// TIA Portal V17 export
// export: Created 2023-02-13T11:16:53.9943503Z, ExportSetting WithDefaults, DisplayName Totally Integrated Automation Portal, DisplayVersion V17, DisplayName TIA Portal Openness, DisplayVersion V17, DisplayName TIA Portal Teamcenter Gateway, DisplayVersion V17, DisplayName TIA Portal Version Control Interface, DisplayVersion V17, DisplayName SINAMICS Startdrive Advanced, DisplayVersion V17, DisplayName SINAMICS Startdrive G130, G150, S120, S150, SINAMICS MV, S210, DisplayVersion V17, DisplayName SINAMICS Startdrive G110M, G120, G120C, G120D, G120P, G115D, DisplayVersion V17, DisplayName STEP 7 Professional, DisplayVersion V17, DisplayName STEP 7 Safety, DisplayVersion V17, DisplayName WinCC Professional, DisplayVersion V17
FUNCTION "Blending" : Void   // FC8, LAD
{ S7_Optimized_Access := 'TRUE' }
VERSION : 0.1
// stored: AutoNumber true, IsIECCheckEnabled false, SetENOAutomatically false, UDAEnableTagReadback false
   VAR_TEMP   // added for the SCL form of the ladder/FBD networks
      _w1 : Bool;
   END_VAR
BEGIN

REGION Network 1
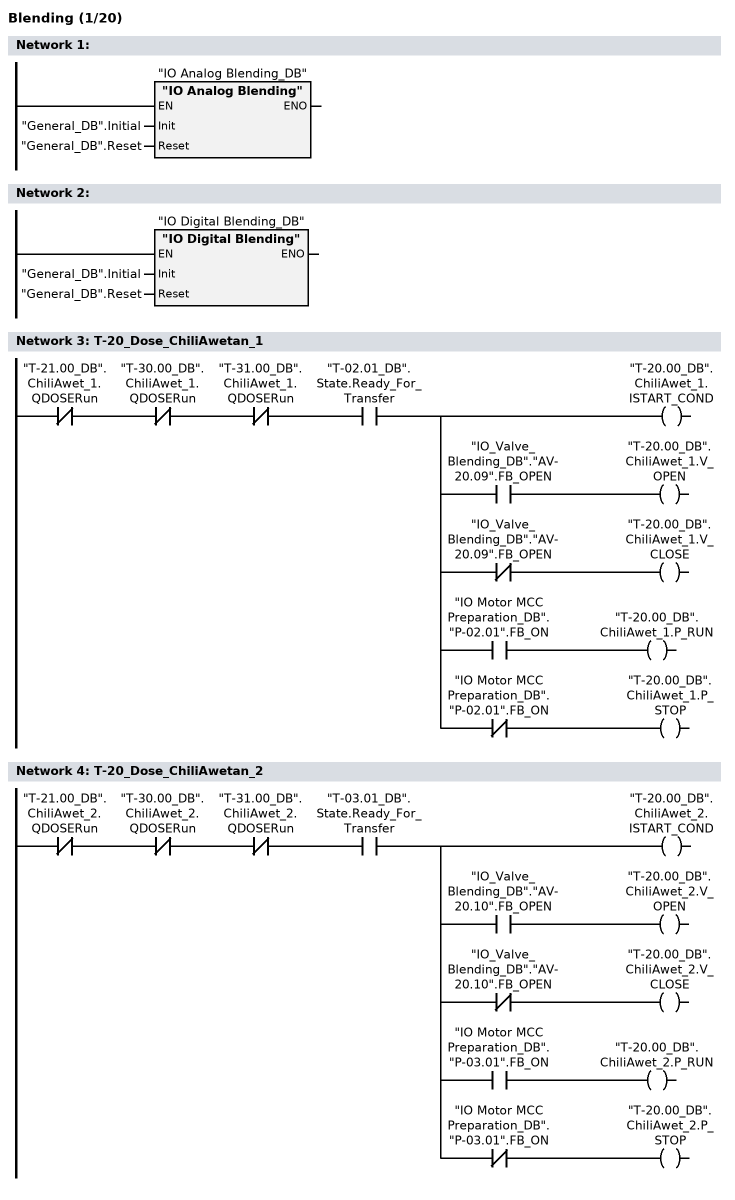
   RUNG wire#powerrail
      "IO Analog Blending_DB"(Init := "General_DB".Initial, Reset := "General_DB".Reset)
   END_RUNG
   // the same network as SCL:
   "IO Analog Blending_DB"(Init := "General_DB".Initial, Reset := "General_DB".Reset);   // "IO Analog Blending"
END_REGION

REGION Network 2
   RUNG wire#powerrail
      "IO Digital Blending_DB"(Init := "General_DB".Initial, Reset := "General_DB".Reset)
   END_RUNG
   // the same network as SCL:
   "IO Digital Blending_DB"(Init := "General_DB".Initial, Reset := "General_DB".Reset);   // "IO Digital Blending"
END_REGION

REGION Network 3: T-20_Dose_ChiliAwetan_1
   RUNG wire#powerrail
      I_Contact( "T-21.00_DB".ChiliAwet_1.QDOSERun )
      I_Contact( "T-30.00_DB".ChiliAwet_1.QDOSERun )
      I_Contact( "T-31.00_DB".ChiliAwet_1.QDOSERun )
      Contact( "T-02.01_DB".State.Ready_For_Transfer )
      wire#w1
      Coil( "T-20.00_DB".ChiliAwet_1.ISTART_COND )
   END_RUNG
   RUNG wire#w1
      Contact( "IO_Valve_Blending_DB"."AV-20.09".FB_OPEN )
      Coil( "T-20.00_DB".ChiliAwet_1.V_OPEN )
   END_RUNG
   RUNG wire#w1
      I_Contact( "IO_Valve_Blending_DB"."AV-20.09".FB_OPEN )
      Coil( "T-20.00_DB".ChiliAwet_1.V_CLOSE )
   END_RUNG
   RUNG wire#w1
      Contact( "IO Motor MCC Preparation_DB"."P-02.01".FB_ON )
      Coil( "T-20.00_DB".ChiliAwet_1.P_RUN )
   END_RUNG
   RUNG wire#w1
      I_Contact( "IO Motor MCC Preparation_DB"."P-02.01".FB_ON )
      Coil( "T-20.00_DB".ChiliAwet_1.P_STOP )
   END_RUNG
   // the same network as SCL:
   "T-20.00_DB".ChiliAwet_1.ISTART_COND := NOT "T-21.00_DB".ChiliAwet_1.QDOSERun AND NOT "T-30.00_DB".ChiliAwet_1.QDOSERun AND NOT "T-31.00_DB".ChiliAwet_1.QDOSERun AND "T-02.01_DB".State.Ready_For_Transfer;
   "T-20.00_DB".ChiliAwet_1.V_OPEN := "T-20.00_DB".ChiliAwet_1.ISTART_COND AND "IO_Valve_Blending_DB"."AV-20.09".FB_OPEN;
   "T-20.00_DB".ChiliAwet_1.V_CLOSE := "T-20.00_DB".ChiliAwet_1.ISTART_COND AND NOT "IO_Valve_Blending_DB"."AV-20.09".FB_OPEN;
   "T-20.00_DB".ChiliAwet_1.P_RUN := "T-20.00_DB".ChiliAwet_1.ISTART_COND AND "IO Motor MCC Preparation_DB"."P-02.01".FB_ON;
   "T-20.00_DB".ChiliAwet_1.P_STOP := "T-20.00_DB".ChiliAwet_1.ISTART_COND AND NOT "IO Motor MCC Preparation_DB"."P-02.01".FB_ON;
END_REGION

REGION Network 4: T-20_Dose_ChiliAwetan_2
   RUNG wire#powerrail
      I_Contact( "T-21.00_DB".ChiliAwet_2.QDOSERun )
      I_Contact( "T-30.00_DB".ChiliAwet_2.QDOSERun )
      I_Contact( "T-31.00_DB".ChiliAwet_2.QDOSERun )
      Contact( "T-03.01_DB".State.Ready_For_Transfer )
      wire#w1
      Coil( "T-20.00_DB".ChiliAwet_2.ISTART_COND )
   END_RUNG
   RUNG wire#w1
      Contact( "IO_Valve_Blending_DB"."AV-20.10".FB_OPEN )
      Coil( "T-20.00_DB".ChiliAwet_2.V_OPEN )
   END_RUNG
   RUNG wire#w1
      I_Contact( "IO_Valve_Blending_DB"."AV-20.10".FB_OPEN )
      Coil( "T-20.00_DB".ChiliAwet_2.V_CLOSE )
   END_RUNG
   RUNG wire#w1
      Contact( "IO Motor MCC Preparation_DB"."P-03.01".FB_ON )
      Coil( "T-20.00_DB".ChiliAwet_2.P_RUN )
   END_RUNG
   RUNG wire#w1
      I_Contact( "IO Motor MCC Preparation_DB"."P-03.01".FB_ON )
      Coil( "T-20.00_DB".ChiliAwet_2.P_STOP )
   END_RUNG
   // the same network as SCL:
   "T-20.00_DB".ChiliAwet_2.ISTART_COND := NOT "T-21.00_DB".ChiliAwet_2.QDOSERun AND NOT "T-30.00_DB".ChiliAwet_2.QDOSERun AND NOT "T-31.00_DB".ChiliAwet_2.QDOSERun AND "T-03.01_DB".State.Ready_For_Transfer;
   "T-20.00_DB".ChiliAwet_2.V_OPEN := "T-20.00_DB".ChiliAwet_2.ISTART_COND AND "IO_Valve_Blending_DB"."AV-20.10".FB_OPEN;
   "T-20.00_DB".ChiliAwet_2.V_CLOSE := "T-20.00_DB".ChiliAwet_2.ISTART_COND AND NOT "IO_Valve_Blending_DB"."AV-20.10".FB_OPEN;
   "T-20.00_DB".ChiliAwet_2.P_RUN := "T-20.00_DB".ChiliAwet_2.ISTART_COND AND "IO Motor MCC Preparation_DB"."P-03.01".FB_ON;
   "T-20.00_DB".ChiliAwet_2.P_STOP := "T-20.00_DB".ChiliAwet_2.ISTART_COND AND NOT "IO Motor MCC Preparation_DB"."P-03.01".FB_ON;
END_REGION

REGION Network 5: T-20_Dose_ChiliAwetan_3
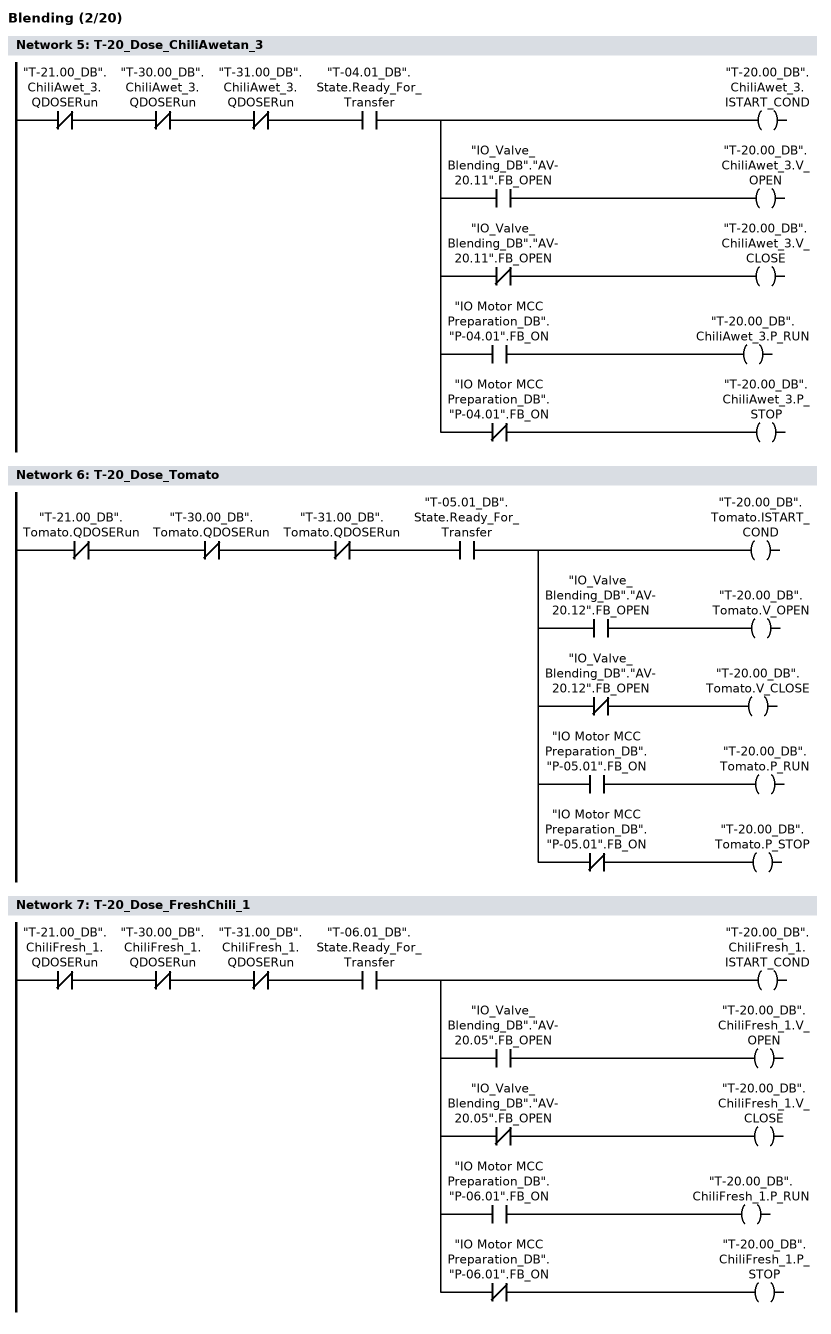
   RUNG wire#powerrail
      I_Contact( "T-21.00_DB".ChiliAwet_3.QDOSERun )
      I_Contact( "T-30.00_DB".ChiliAwet_3.QDOSERun )
      I_Contact( "T-31.00_DB".ChiliAwet_3.QDOSERun )
      Contact( "T-04.01_DB".State.Ready_For_Transfer )
      wire#w1
      Coil( "T-20.00_DB".ChiliAwet_3.ISTART_COND )
   END_RUNG
   RUNG wire#w1
      Contact( "IO_Valve_Blending_DB"."AV-20.11".FB_OPEN )
      Coil( "T-20.00_DB".ChiliAwet_3.V_OPEN )
   END_RUNG
   RUNG wire#w1
      I_Contact( "IO_Valve_Blending_DB"."AV-20.11".FB_OPEN )
      Coil( "T-20.00_DB".ChiliAwet_3.V_CLOSE )
   END_RUNG
   RUNG wire#w1
      Contact( "IO Motor MCC Preparation_DB"."P-04.01".FB_ON )
      Coil( "T-20.00_DB".ChiliAwet_3.P_RUN )
   END_RUNG
   RUNG wire#w1
      I_Contact( "IO Motor MCC Preparation_DB"."P-04.01".FB_ON )
      Coil( "T-20.00_DB".ChiliAwet_3.P_STOP )
   END_RUNG
   // the same network as SCL:
   "T-20.00_DB".ChiliAwet_3.ISTART_COND := NOT "T-21.00_DB".ChiliAwet_3.QDOSERun AND NOT "T-30.00_DB".ChiliAwet_3.QDOSERun AND NOT "T-31.00_DB".ChiliAwet_3.QDOSERun AND "T-04.01_DB".State.Ready_For_Transfer;
   "T-20.00_DB".ChiliAwet_3.V_OPEN := "T-20.00_DB".ChiliAwet_3.ISTART_COND AND "IO_Valve_Blending_DB"."AV-20.11".FB_OPEN;
   "T-20.00_DB".ChiliAwet_3.V_CLOSE := "T-20.00_DB".ChiliAwet_3.ISTART_COND AND NOT "IO_Valve_Blending_DB"."AV-20.11".FB_OPEN;
   "T-20.00_DB".ChiliAwet_3.P_RUN := "T-20.00_DB".ChiliAwet_3.ISTART_COND AND "IO Motor MCC Preparation_DB"."P-04.01".FB_ON;
   "T-20.00_DB".ChiliAwet_3.P_STOP := "T-20.00_DB".ChiliAwet_3.ISTART_COND AND NOT "IO Motor MCC Preparation_DB"."P-04.01".FB_ON;
END_REGION

REGION Network 6: T-20_Dose_Tomato
   RUNG wire#powerrail
      I_Contact( "T-21.00_DB".Tomato.QDOSERun )
      I_Contact( "T-30.00_DB".Tomato.QDOSERun )
      I_Contact( "T-31.00_DB".Tomato.QDOSERun )
      Contact( "T-05.01_DB".State.Ready_For_Transfer )
      wire#w1
      Coil( "T-20.00_DB".Tomato.ISTART_COND )
   END_RUNG
   RUNG wire#w1
      Contact( "IO_Valve_Blending_DB"."AV-20.12".FB_OPEN )
      Coil( "T-20.00_DB".Tomato.V_OPEN )
   END_RUNG
   RUNG wire#w1
      I_Contact( "IO_Valve_Blending_DB"."AV-20.12".FB_OPEN )
      Coil( "T-20.00_DB".Tomato.V_CLOSE )
   END_RUNG
   RUNG wire#w1
      Contact( "IO Motor MCC Preparation_DB"."P-05.01".FB_ON )
      Coil( "T-20.00_DB".Tomato.P_RUN )
   END_RUNG
   RUNG wire#w1
      I_Contact( "IO Motor MCC Preparation_DB"."P-05.01".FB_ON )
      Coil( "T-20.00_DB".Tomato.P_STOP )
   END_RUNG
   // the same network as SCL:
   "T-20.00_DB".Tomato.ISTART_COND := NOT "T-21.00_DB".Tomato.QDOSERun AND NOT "T-30.00_DB".Tomato.QDOSERun AND NOT "T-31.00_DB".Tomato.QDOSERun AND "T-05.01_DB".State.Ready_For_Transfer;
   "T-20.00_DB".Tomato.V_OPEN := "T-20.00_DB".Tomato.ISTART_COND AND "IO_Valve_Blending_DB"."AV-20.12".FB_OPEN;
   "T-20.00_DB".Tomato.V_CLOSE := "T-20.00_DB".Tomato.ISTART_COND AND NOT "IO_Valve_Blending_DB"."AV-20.12".FB_OPEN;
   "T-20.00_DB".Tomato.P_RUN := "T-20.00_DB".Tomato.ISTART_COND AND "IO Motor MCC Preparation_DB"."P-05.01".FB_ON;
   "T-20.00_DB".Tomato.P_STOP := "T-20.00_DB".Tomato.ISTART_COND AND NOT "IO Motor MCC Preparation_DB"."P-05.01".FB_ON;
END_REGION

REGION Network 7: T-20_Dose_FreshChili_1
   RUNG wire#powerrail
      I_Contact( "T-21.00_DB".ChiliFresh_1.QDOSERun )
      I_Contact( "T-30.00_DB".ChiliFresh_1.QDOSERun )
      I_Contact( "T-31.00_DB".ChiliFresh_1.QDOSERun )
      Contact( "T-06.01_DB".State.Ready_For_Transfer )
      wire#w1
      Coil( "T-20.00_DB".ChiliFresh_1.ISTART_COND )
   END_RUNG
   RUNG wire#w1
      Contact( "IO_Valve_Blending_DB"."AV-20.05".FB_OPEN )
      Coil( "T-20.00_DB".ChiliFresh_1.V_OPEN )
   END_RUNG
   RUNG wire#w1
      I_Contact( "IO_Valve_Blending_DB"."AV-20.05".FB_OPEN )
      Coil( "T-20.00_DB".ChiliFresh_1.V_CLOSE )
   END_RUNG
   RUNG wire#w1
      Contact( "IO Motor MCC Preparation_DB"."P-06.01".FB_ON )
      Coil( "T-20.00_DB".ChiliFresh_1.P_RUN )
   END_RUNG
   RUNG wire#w1
      I_Contact( "IO Motor MCC Preparation_DB"."P-06.01".FB_ON )
      Coil( "T-20.00_DB".ChiliFresh_1.P_STOP )
   END_RUNG
   // the same network as SCL:
   "T-20.00_DB".ChiliFresh_1.ISTART_COND := NOT "T-21.00_DB".ChiliFresh_1.QDOSERun AND NOT "T-30.00_DB".ChiliFresh_1.QDOSERun AND NOT "T-31.00_DB".ChiliFresh_1.QDOSERun AND "T-06.01_DB".State.Ready_For_Transfer;
   "T-20.00_DB".ChiliFresh_1.V_OPEN := "T-20.00_DB".ChiliFresh_1.ISTART_COND AND "IO_Valve_Blending_DB"."AV-20.05".FB_OPEN;
   "T-20.00_DB".ChiliFresh_1.V_CLOSE := "T-20.00_DB".ChiliFresh_1.ISTART_COND AND NOT "IO_Valve_Blending_DB"."AV-20.05".FB_OPEN;
   "T-20.00_DB".ChiliFresh_1.P_RUN := "T-20.00_DB".ChiliFresh_1.ISTART_COND AND "IO Motor MCC Preparation_DB"."P-06.01".FB_ON;
   "T-20.00_DB".ChiliFresh_1.P_STOP := "T-20.00_DB".ChiliFresh_1.ISTART_COND AND NOT "IO Motor MCC Preparation_DB"."P-06.01".FB_ON;
END_REGION

REGION Network 8: T-20_Dose_FreshChili_2
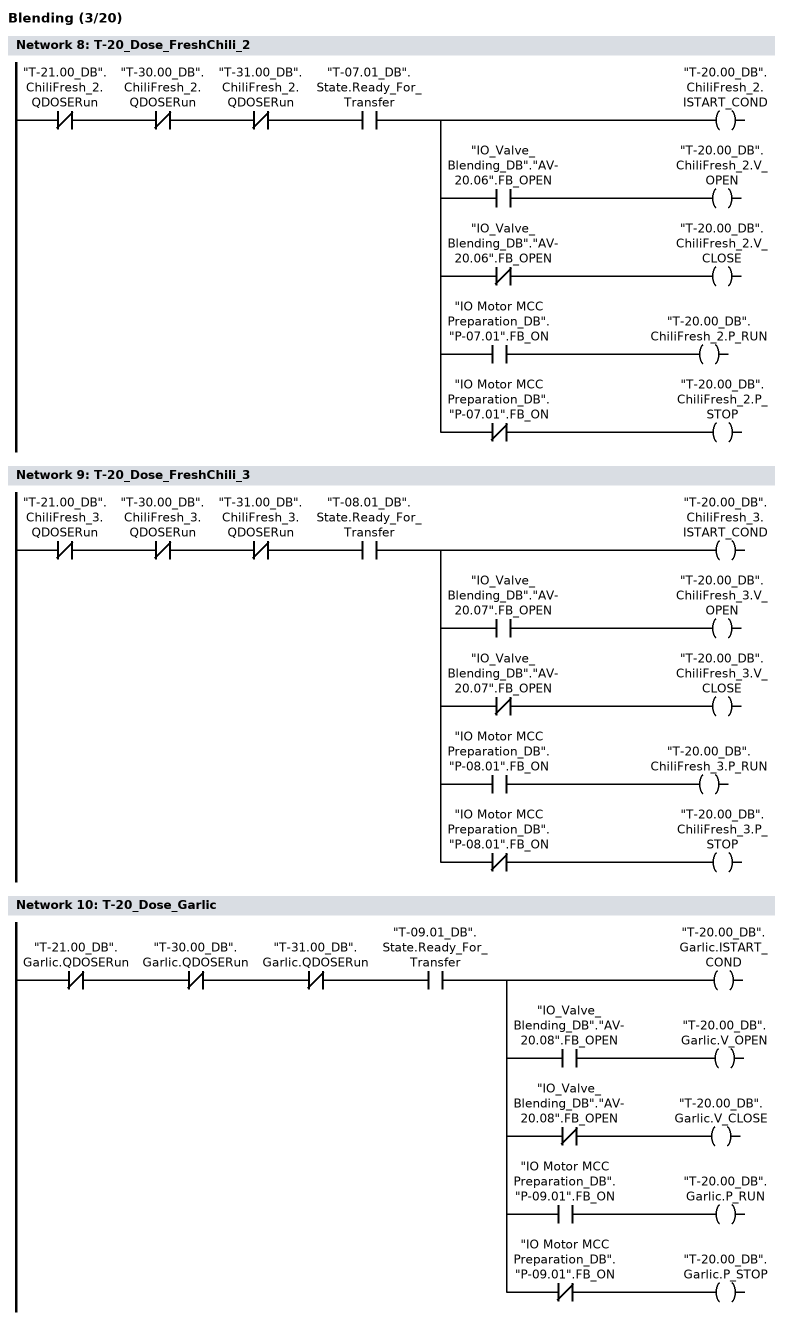
   RUNG wire#powerrail
      I_Contact( "T-21.00_DB".ChiliFresh_2.QDOSERun )
      I_Contact( "T-30.00_DB".ChiliFresh_2.QDOSERun )
      I_Contact( "T-31.00_DB".ChiliFresh_2.QDOSERun )
      Contact( "T-07.01_DB".State.Ready_For_Transfer )
      wire#w1
      Coil( "T-20.00_DB".ChiliFresh_2.ISTART_COND )
   END_RUNG
   RUNG wire#w1
      Contact( "IO_Valve_Blending_DB"."AV-20.06".FB_OPEN )
      Coil( "T-20.00_DB".ChiliFresh_2.V_OPEN )
   END_RUNG
   RUNG wire#w1
      I_Contact( "IO_Valve_Blending_DB"."AV-20.06".FB_OPEN )
      Coil( "T-20.00_DB".ChiliFresh_2.V_CLOSE )
   END_RUNG
   RUNG wire#w1
      Contact( "IO Motor MCC Preparation_DB"."P-07.01".FB_ON )
      Coil( "T-20.00_DB".ChiliFresh_2.P_RUN )
   END_RUNG
   RUNG wire#w1
      I_Contact( "IO Motor MCC Preparation_DB"."P-07.01".FB_ON )
      Coil( "T-20.00_DB".ChiliFresh_2.P_STOP )
   END_RUNG
   // the same network as SCL:
   "T-20.00_DB".ChiliFresh_2.ISTART_COND := NOT "T-21.00_DB".ChiliFresh_2.QDOSERun AND NOT "T-30.00_DB".ChiliFresh_2.QDOSERun AND NOT "T-31.00_DB".ChiliFresh_2.QDOSERun AND "T-07.01_DB".State.Ready_For_Transfer;
   "T-20.00_DB".ChiliFresh_2.V_OPEN := "T-20.00_DB".ChiliFresh_2.ISTART_COND AND "IO_Valve_Blending_DB"."AV-20.06".FB_OPEN;
   "T-20.00_DB".ChiliFresh_2.V_CLOSE := "T-20.00_DB".ChiliFresh_2.ISTART_COND AND NOT "IO_Valve_Blending_DB"."AV-20.06".FB_OPEN;
   "T-20.00_DB".ChiliFresh_2.P_RUN := "T-20.00_DB".ChiliFresh_2.ISTART_COND AND "IO Motor MCC Preparation_DB"."P-07.01".FB_ON;
   "T-20.00_DB".ChiliFresh_2.P_STOP := "T-20.00_DB".ChiliFresh_2.ISTART_COND AND NOT "IO Motor MCC Preparation_DB"."P-07.01".FB_ON;
END_REGION

REGION Network 9: T-20_Dose_FreshChili_3
   RUNG wire#powerrail
      I_Contact( "T-21.00_DB".ChiliFresh_3.QDOSERun )
      I_Contact( "T-30.00_DB".ChiliFresh_3.QDOSERun )
      I_Contact( "T-31.00_DB".ChiliFresh_3.QDOSERun )
      Contact( "T-08.01_DB".State.Ready_For_Transfer )
      wire#w1
      Coil( "T-20.00_DB".ChiliFresh_3.ISTART_COND )
   END_RUNG
   RUNG wire#w1
      Contact( "IO_Valve_Blending_DB"."AV-20.07".FB_OPEN )
      Coil( "T-20.00_DB".ChiliFresh_3.V_OPEN )
   END_RUNG
   RUNG wire#w1
      I_Contact( "IO_Valve_Blending_DB"."AV-20.07".FB_OPEN )
      Coil( "T-20.00_DB".ChiliFresh_3.V_CLOSE )
   END_RUNG
   RUNG wire#w1
      Contact( "IO Motor MCC Preparation_DB"."P-08.01".FB_ON )
      Coil( "T-20.00_DB".ChiliFresh_3.P_RUN )
   END_RUNG
   RUNG wire#w1
      I_Contact( "IO Motor MCC Preparation_DB"."P-08.01".FB_ON )
      Coil( "T-20.00_DB".ChiliFresh_3.P_STOP )
   END_RUNG
   // the same network as SCL:
   "T-20.00_DB".ChiliFresh_3.ISTART_COND := NOT "T-21.00_DB".ChiliFresh_3.QDOSERun AND NOT "T-30.00_DB".ChiliFresh_3.QDOSERun AND NOT "T-31.00_DB".ChiliFresh_3.QDOSERun AND "T-08.01_DB".State.Ready_For_Transfer;
   "T-20.00_DB".ChiliFresh_3.V_OPEN := "T-20.00_DB".ChiliFresh_3.ISTART_COND AND "IO_Valve_Blending_DB"."AV-20.07".FB_OPEN;
   "T-20.00_DB".ChiliFresh_3.V_CLOSE := "T-20.00_DB".ChiliFresh_3.ISTART_COND AND NOT "IO_Valve_Blending_DB"."AV-20.07".FB_OPEN;
   "T-20.00_DB".ChiliFresh_3.P_RUN := "T-20.00_DB".ChiliFresh_3.ISTART_COND AND "IO Motor MCC Preparation_DB"."P-08.01".FB_ON;
   "T-20.00_DB".ChiliFresh_3.P_STOP := "T-20.00_DB".ChiliFresh_3.ISTART_COND AND NOT "IO Motor MCC Preparation_DB"."P-08.01".FB_ON;
END_REGION

REGION Network 10: T-20_Dose_Garlic
   RUNG wire#powerrail
      I_Contact( "T-21.00_DB".Garlic.QDOSERun )
      I_Contact( "T-30.00_DB".Garlic.QDOSERun )
      I_Contact( "T-31.00_DB".Garlic.QDOSERun )
      Contact( "T-09.01_DB".State.Ready_For_Transfer )
      wire#w1
      Coil( "T-20.00_DB".Garlic.ISTART_COND )
   END_RUNG
   RUNG wire#w1
      Contact( "IO_Valve_Blending_DB"."AV-20.08".FB_OPEN )
      Coil( "T-20.00_DB".Garlic.V_OPEN )
   END_RUNG
   RUNG wire#w1
      I_Contact( "IO_Valve_Blending_DB"."AV-20.08".FB_OPEN )
      Coil( "T-20.00_DB".Garlic.V_CLOSE )
   END_RUNG
   RUNG wire#w1
      Contact( "IO Motor MCC Preparation_DB"."P-09.01".FB_ON )
      Coil( "T-20.00_DB".Garlic.P_RUN )
   END_RUNG
   RUNG wire#w1
      I_Contact( "IO Motor MCC Preparation_DB"."P-09.01".FB_ON )
      Coil( "T-20.00_DB".Garlic.P_STOP )
   END_RUNG
   // the same network as SCL:
   "T-20.00_DB".Garlic.ISTART_COND := NOT "T-21.00_DB".Garlic.QDOSERun AND NOT "T-30.00_DB".Garlic.QDOSERun AND NOT "T-31.00_DB".Garlic.QDOSERun AND "T-09.01_DB".State.Ready_For_Transfer;
   "T-20.00_DB".Garlic.V_OPEN := "T-20.00_DB".Garlic.ISTART_COND AND "IO_Valve_Blending_DB"."AV-20.08".FB_OPEN;
   "T-20.00_DB".Garlic.V_CLOSE := "T-20.00_DB".Garlic.ISTART_COND AND NOT "IO_Valve_Blending_DB"."AV-20.08".FB_OPEN;
   "T-20.00_DB".Garlic.P_RUN := "T-20.00_DB".Garlic.ISTART_COND AND "IO Motor MCC Preparation_DB"."P-09.01".FB_ON;
   "T-20.00_DB".Garlic.P_STOP := "T-20.00_DB".Garlic.ISTART_COND AND NOT "IO Motor MCC Preparation_DB"."P-09.01".FB_ON;
END_REGION

REGION Network 11: T-20_Dose_Vinegar
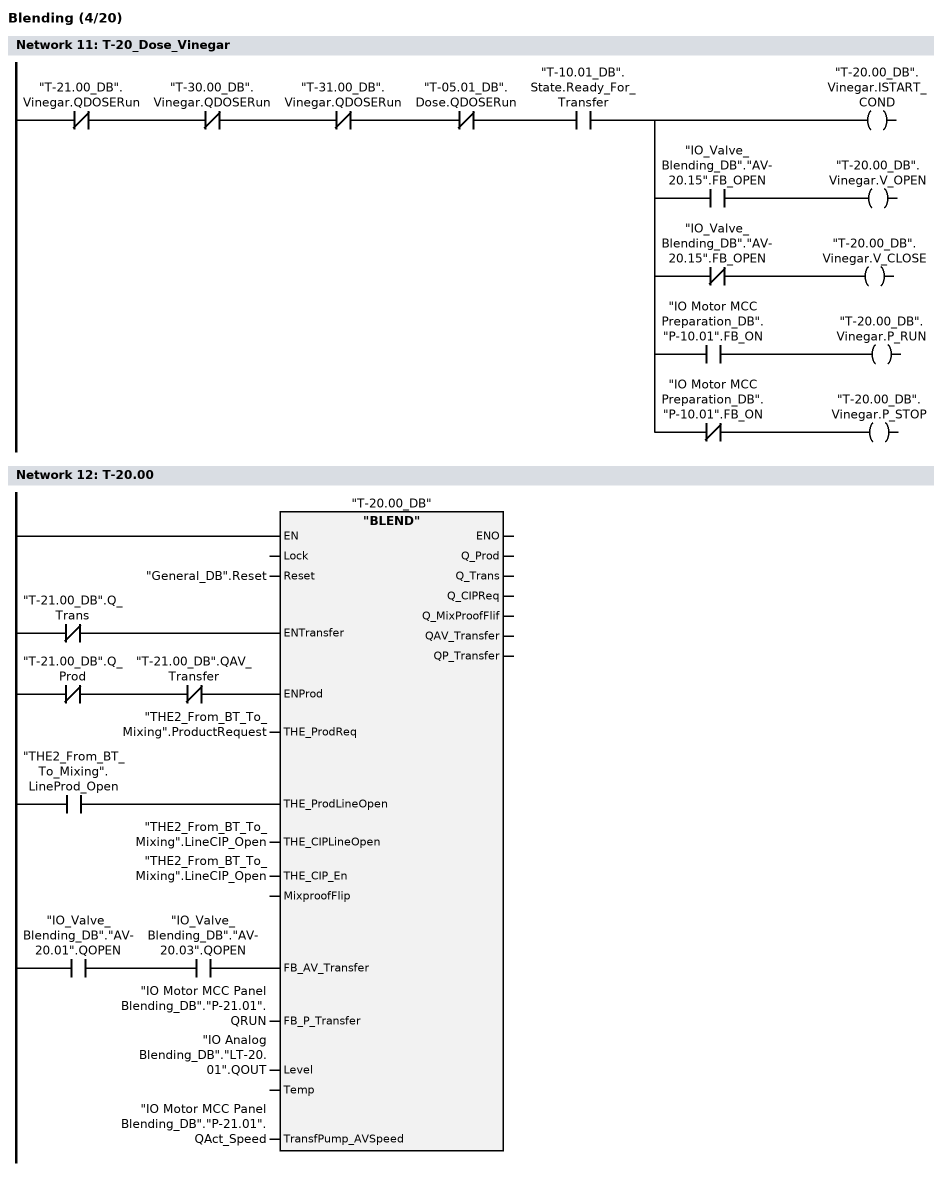
   RUNG wire#powerrail
      I_Contact( "T-21.00_DB".Vinegar.QDOSERun )
      I_Contact( "T-30.00_DB".Vinegar.QDOSERun )
      I_Contact( "T-31.00_DB".Vinegar.QDOSERun )
      I_Contact( "T-05.01_DB".Dose.QDOSERun )
      Contact( "T-10.01_DB".State.Ready_For_Transfer )
      wire#w1
      Coil( "T-20.00_DB".Vinegar.ISTART_COND )
   END_RUNG
   RUNG wire#w1
      Contact( "IO_Valve_Blending_DB"."AV-20.15".FB_OPEN )
      Coil( "T-20.00_DB".Vinegar.V_OPEN )
   END_RUNG
   RUNG wire#w1
      I_Contact( "IO_Valve_Blending_DB"."AV-20.15".FB_OPEN )
      Coil( "T-20.00_DB".Vinegar.V_CLOSE )
   END_RUNG
   RUNG wire#w1
      Contact( "IO Motor MCC Preparation_DB"."P-10.01".FB_ON )
      Coil( "T-20.00_DB".Vinegar.P_RUN )
   END_RUNG
   RUNG wire#w1
      I_Contact( "IO Motor MCC Preparation_DB"."P-10.01".FB_ON )
      Coil( "T-20.00_DB".Vinegar.P_STOP )
   END_RUNG
   // the same network as SCL:
   "T-20.00_DB".Vinegar.ISTART_COND := NOT "T-21.00_DB".Vinegar.QDOSERun AND NOT "T-30.00_DB".Vinegar.QDOSERun AND NOT "T-31.00_DB".Vinegar.QDOSERun AND NOT "T-05.01_DB".Dose.QDOSERun AND "T-10.01_DB".State.Ready_For_Transfer;
   "T-20.00_DB".Vinegar.V_OPEN := "T-20.00_DB".Vinegar.ISTART_COND AND "IO_Valve_Blending_DB"."AV-20.15".FB_OPEN;
   "T-20.00_DB".Vinegar.V_CLOSE := "T-20.00_DB".Vinegar.ISTART_COND AND NOT "IO_Valve_Blending_DB"."AV-20.15".FB_OPEN;
   "T-20.00_DB".Vinegar.P_RUN := "T-20.00_DB".Vinegar.ISTART_COND AND "IO Motor MCC Preparation_DB"."P-10.01".FB_ON;
   "T-20.00_DB".Vinegar.P_STOP := "T-20.00_DB".Vinegar.ISTART_COND AND NOT "IO Motor MCC Preparation_DB"."P-10.01".FB_ON;
END_REGION

REGION Network 12: T-20.00
   RUNG wire#powerrail
      "T-20.00_DB"(ENTransfer := wire#w1, ENProd := wire#w2, THE_ProdLineOpen := wire#w3, FB_AV_Transfer := wire#w4, Lock :=, Reset := "General_DB".Reset, THE_ProdReq := "THE2_From_BT_To_Mixing".ProductRequest, THE_CIPLineOpen := "THE2_From_BT_To_Mixing".LineCIP_Open, THE_CIP_En := "THE2_From_BT_To_Mixing".LineCIP_Open, MixproofFlip :=, FB_P_Transfer := "IO Motor MCC Panel Blending_DB"."P-21.01".QRUN, Level := "IO Analog Blending_DB"."LT-20.01".QOUT, Temp :=, TransfPump_AVSpeed := "IO Motor MCC Panel Blending_DB"."P-21.01".QAct_Speed, Q_Prod =>, Q_Trans =>, Q_CIPReq =>, Q_MixProofFlif =>, QAV_Transfer =>, QP_Transfer =>)
   END_RUNG
   RUNG wire#powerrail
      I_Contact( "T-21.00_DB".Q_Trans )
   END_RUNG wire#w1
   RUNG wire#powerrail
      I_Contact( "T-21.00_DB".Q_Prod )
      I_Contact( "T-21.00_DB".QAV_Transfer )
   END_RUNG wire#w2
   RUNG wire#powerrail
      Contact( "THE2_From_BT_To_Mixing".LineProd_Open )
   END_RUNG wire#w3
   RUNG wire#powerrail
      Contact( "IO_Valve_Blending_DB"."AV-20.01".QOPEN )
      Contact( "IO_Valve_Blending_DB"."AV-20.03".QOPEN )
   END_RUNG wire#w4
   // the same network as SCL:
   "T-20.00_DB"(Reset := "General_DB".Reset,   // "BLEND"
                ENTransfer := NOT "T-21.00_DB".Q_Trans,
                ENProd := NOT "T-21.00_DB".Q_Prod AND NOT "T-21.00_DB".QAV_Transfer,
                THE_ProdReq := "THE2_From_BT_To_Mixing".ProductRequest,
                THE_ProdLineOpen := "THE2_From_BT_To_Mixing".LineProd_Open,
                THE_CIPLineOpen := "THE2_From_BT_To_Mixing".LineCIP_Open,
                THE_CIP_En := "THE2_From_BT_To_Mixing".LineCIP_Open,
                FB_AV_Transfer := "IO_Valve_Blending_DB"."AV-20.01".QOPEN AND "IO_Valve_Blending_DB"."AV-20.03".QOPEN,
                FB_P_Transfer := "IO Motor MCC Panel Blending_DB"."P-21.01".QRUN,
                Level := "IO Analog Blending_DB"."LT-20.01".QOUT,
                TransfPump_AVSpeed := "IO Motor MCC Panel Blending_DB"."P-21.01".QAct_Speed);
END_REGION

REGION Network 14: T-21_Dose_ChiliAwetan_1
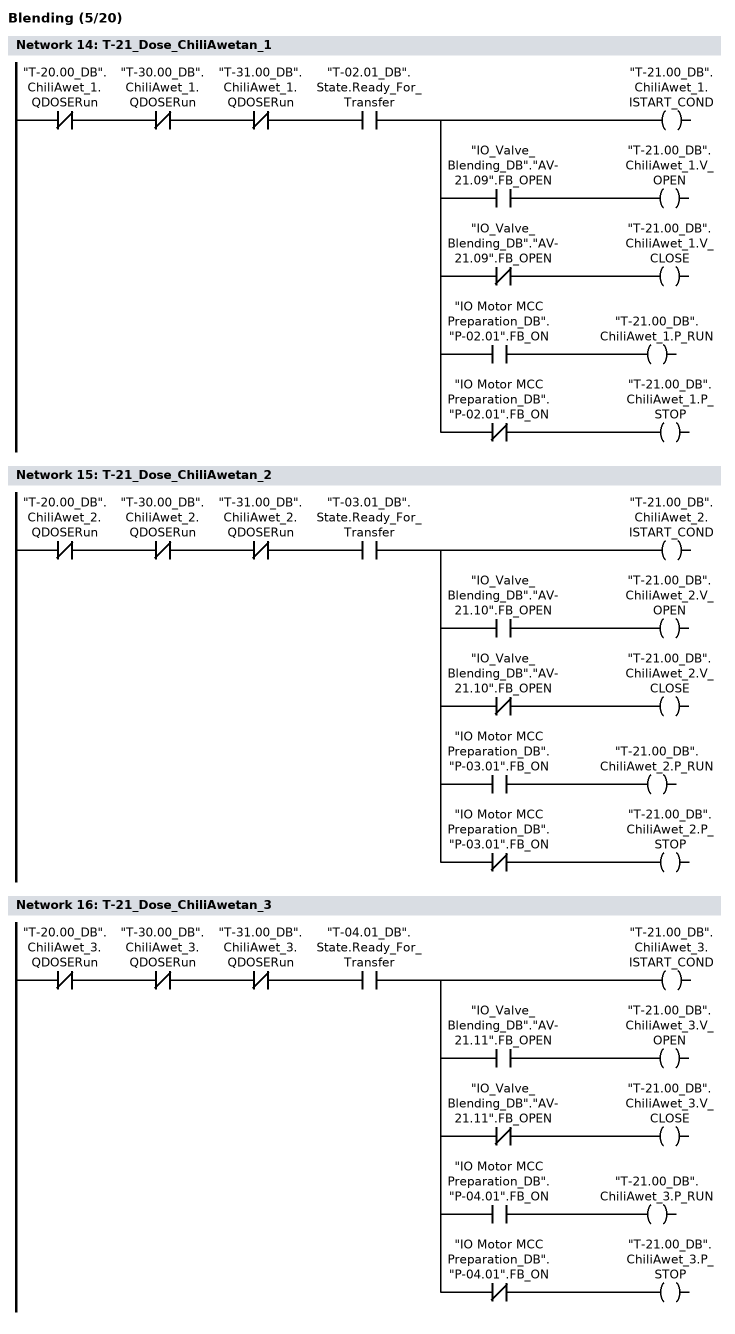
   RUNG wire#powerrail
      I_Contact( "T-20.00_DB".ChiliAwet_1.QDOSERun )
      I_Contact( "T-30.00_DB".ChiliAwet_1.QDOSERun )
      I_Contact( "T-31.00_DB".ChiliAwet_1.QDOSERun )
      Contact( "T-02.01_DB".State.Ready_For_Transfer )
      wire#w1
      Coil( "T-21.00_DB".ChiliAwet_1.ISTART_COND )
   END_RUNG
   RUNG wire#w1
      Contact( "IO_Valve_Blending_DB"."AV-21.09".FB_OPEN )
      Coil( "T-21.00_DB".ChiliAwet_1.V_OPEN )
   END_RUNG
   RUNG wire#w1
      I_Contact( "IO_Valve_Blending_DB"."AV-21.09".FB_OPEN )
      Coil( "T-21.00_DB".ChiliAwet_1.V_CLOSE )
   END_RUNG
   RUNG wire#w1
      Contact( "IO Motor MCC Preparation_DB"."P-02.01".FB_ON )
      Coil( "T-21.00_DB".ChiliAwet_1.P_RUN )
   END_RUNG
   RUNG wire#w1
      I_Contact( "IO Motor MCC Preparation_DB"."P-02.01".FB_ON )
      Coil( "T-21.00_DB".ChiliAwet_1.P_STOP )
   END_RUNG
   // the same network as SCL:
   "T-21.00_DB".ChiliAwet_1.ISTART_COND := NOT "T-20.00_DB".ChiliAwet_1.QDOSERun AND NOT "T-30.00_DB".ChiliAwet_1.QDOSERun AND NOT "T-31.00_DB".ChiliAwet_1.QDOSERun AND "T-02.01_DB".State.Ready_For_Transfer;
   "T-21.00_DB".ChiliAwet_1.V_OPEN := "T-21.00_DB".ChiliAwet_1.ISTART_COND AND "IO_Valve_Blending_DB"."AV-21.09".FB_OPEN;
   "T-21.00_DB".ChiliAwet_1.V_CLOSE := "T-21.00_DB".ChiliAwet_1.ISTART_COND AND NOT "IO_Valve_Blending_DB"."AV-21.09".FB_OPEN;
   "T-21.00_DB".ChiliAwet_1.P_RUN := "T-21.00_DB".ChiliAwet_1.ISTART_COND AND "IO Motor MCC Preparation_DB"."P-02.01".FB_ON;
   "T-21.00_DB".ChiliAwet_1.P_STOP := "T-21.00_DB".ChiliAwet_1.ISTART_COND AND NOT "IO Motor MCC Preparation_DB"."P-02.01".FB_ON;
END_REGION

REGION Network 15: T-21_Dose_ChiliAwetan_2
   RUNG wire#powerrail
      I_Contact( "T-20.00_DB".ChiliAwet_2.QDOSERun )
      I_Contact( "T-30.00_DB".ChiliAwet_2.QDOSERun )
      I_Contact( "T-31.00_DB".ChiliAwet_2.QDOSERun )
      Contact( "T-03.01_DB".State.Ready_For_Transfer )
      wire#w1
      Coil( "T-21.00_DB".ChiliAwet_2.ISTART_COND )
   END_RUNG
   RUNG wire#w1
      Contact( "IO_Valve_Blending_DB"."AV-21.10".FB_OPEN )
      Coil( "T-21.00_DB".ChiliAwet_2.V_OPEN )
   END_RUNG
   RUNG wire#w1
      I_Contact( "IO_Valve_Blending_DB"."AV-21.10".FB_OPEN )
      Coil( "T-21.00_DB".ChiliAwet_2.V_CLOSE )
   END_RUNG
   RUNG wire#w1
      Contact( "IO Motor MCC Preparation_DB"."P-03.01".FB_ON )
      Coil( "T-21.00_DB".ChiliAwet_2.P_RUN )
   END_RUNG
   RUNG wire#w1
      I_Contact( "IO Motor MCC Preparation_DB"."P-03.01".FB_ON )
      Coil( "T-21.00_DB".ChiliAwet_2.P_STOP )
   END_RUNG
   // the same network as SCL:
   "T-21.00_DB".ChiliAwet_2.ISTART_COND := NOT "T-20.00_DB".ChiliAwet_2.QDOSERun AND NOT "T-30.00_DB".ChiliAwet_2.QDOSERun AND NOT "T-31.00_DB".ChiliAwet_2.QDOSERun AND "T-03.01_DB".State.Ready_For_Transfer;
   "T-21.00_DB".ChiliAwet_2.V_OPEN := "T-21.00_DB".ChiliAwet_2.ISTART_COND AND "IO_Valve_Blending_DB"."AV-21.10".FB_OPEN;
   "T-21.00_DB".ChiliAwet_2.V_CLOSE := "T-21.00_DB".ChiliAwet_2.ISTART_COND AND NOT "IO_Valve_Blending_DB"."AV-21.10".FB_OPEN;
   "T-21.00_DB".ChiliAwet_2.P_RUN := "T-21.00_DB".ChiliAwet_2.ISTART_COND AND "IO Motor MCC Preparation_DB"."P-03.01".FB_ON;
   "T-21.00_DB".ChiliAwet_2.P_STOP := "T-21.00_DB".ChiliAwet_2.ISTART_COND AND NOT "IO Motor MCC Preparation_DB"."P-03.01".FB_ON;
END_REGION

REGION Network 16: T-21_Dose_ChiliAwetan_3
   RUNG wire#powerrail
      I_Contact( "T-20.00_DB".ChiliAwet_3.QDOSERun )
      I_Contact( "T-30.00_DB".ChiliAwet_3.QDOSERun )
      I_Contact( "T-31.00_DB".ChiliAwet_3.QDOSERun )
      Contact( "T-04.01_DB".State.Ready_For_Transfer )
      wire#w1
      Coil( "T-21.00_DB".ChiliAwet_3.ISTART_COND )
   END_RUNG
   RUNG wire#w1
      Contact( "IO_Valve_Blending_DB"."AV-21.11".FB_OPEN )
      Coil( "T-21.00_DB".ChiliAwet_3.V_OPEN )
   END_RUNG
   RUNG wire#w1
      I_Contact( "IO_Valve_Blending_DB"."AV-21.11".FB_OPEN )
      Coil( "T-21.00_DB".ChiliAwet_3.V_CLOSE )
   END_RUNG
   RUNG wire#w1
      Contact( "IO Motor MCC Preparation_DB"."P-04.01".FB_ON )
      Coil( "T-21.00_DB".ChiliAwet_3.P_RUN )
   END_RUNG
   RUNG wire#w1
      I_Contact( "IO Motor MCC Preparation_DB"."P-04.01".FB_ON )
      Coil( "T-21.00_DB".ChiliAwet_3.P_STOP )
   END_RUNG
   // the same network as SCL:
   "T-21.00_DB".ChiliAwet_3.ISTART_COND := NOT "T-20.00_DB".ChiliAwet_3.QDOSERun AND NOT "T-30.00_DB".ChiliAwet_3.QDOSERun AND NOT "T-31.00_DB".ChiliAwet_3.QDOSERun AND "T-04.01_DB".State.Ready_For_Transfer;
   "T-21.00_DB".ChiliAwet_3.V_OPEN := "T-21.00_DB".ChiliAwet_3.ISTART_COND AND "IO_Valve_Blending_DB"."AV-21.11".FB_OPEN;
   "T-21.00_DB".ChiliAwet_3.V_CLOSE := "T-21.00_DB".ChiliAwet_3.ISTART_COND AND NOT "IO_Valve_Blending_DB"."AV-21.11".FB_OPEN;
   "T-21.00_DB".ChiliAwet_3.P_RUN := "T-21.00_DB".ChiliAwet_3.ISTART_COND AND "IO Motor MCC Preparation_DB"."P-04.01".FB_ON;
   "T-21.00_DB".ChiliAwet_3.P_STOP := "T-21.00_DB".ChiliAwet_3.ISTART_COND AND NOT "IO Motor MCC Preparation_DB"."P-04.01".FB_ON;
END_REGION

REGION Network 17: T-21_Dose_Tomato
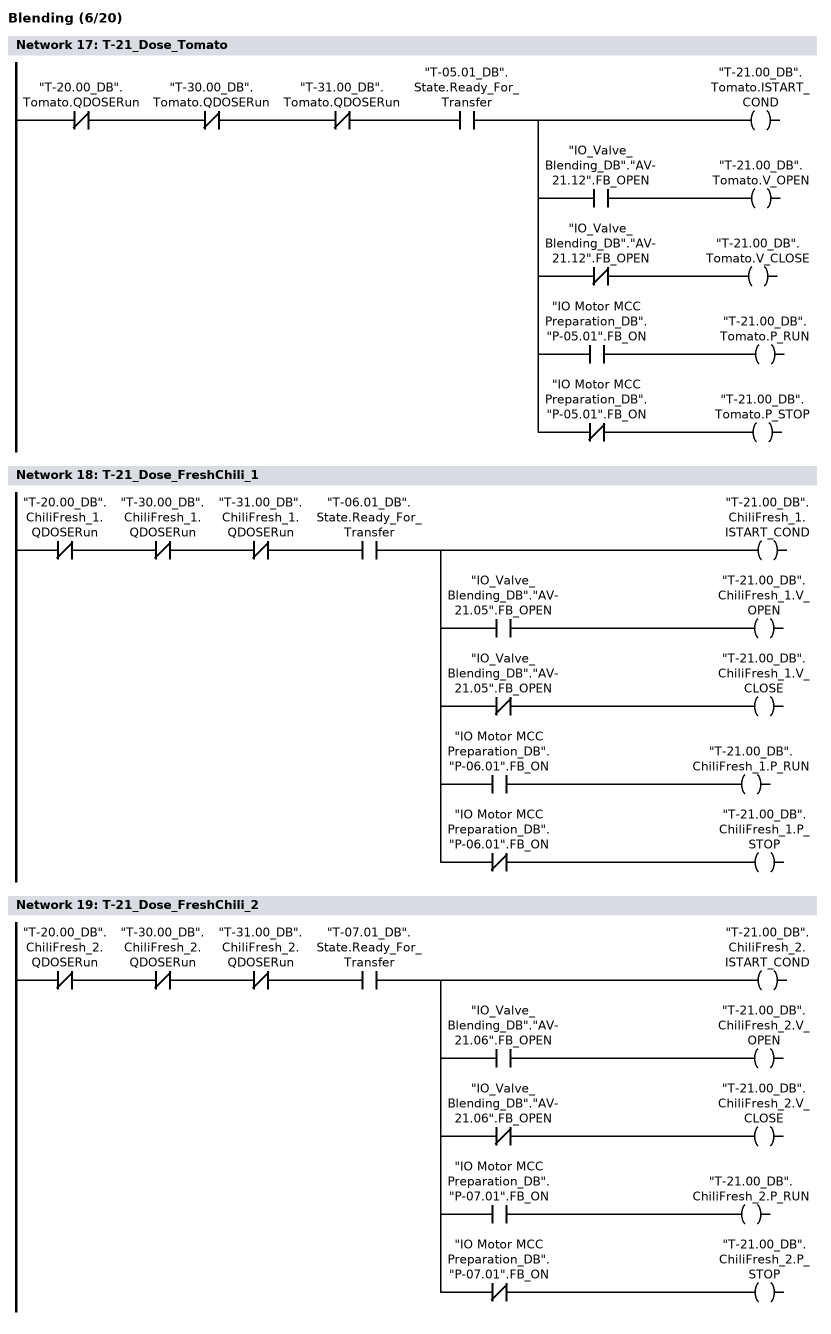
   RUNG wire#powerrail
      I_Contact( "T-20.00_DB".Tomato.QDOSERun )
      I_Contact( "T-30.00_DB".Tomato.QDOSERun )
      I_Contact( "T-31.00_DB".Tomato.QDOSERun )
      Contact( "T-05.01_DB".State.Ready_For_Transfer )
      wire#w1
      Coil( "T-21.00_DB".Tomato.ISTART_COND )
   END_RUNG
   RUNG wire#w1
      Contact( "IO_Valve_Blending_DB"."AV-21.12".FB_OPEN )
      Coil( "T-21.00_DB".Tomato.V_OPEN )
   END_RUNG
   RUNG wire#w1
      I_Contact( "IO_Valve_Blending_DB"."AV-21.12".FB_OPEN )
      Coil( "T-21.00_DB".Tomato.V_CLOSE )
   END_RUNG
   RUNG wire#w1
      Contact( "IO Motor MCC Preparation_DB"."P-05.01".FB_ON )
      Coil( "T-21.00_DB".Tomato.P_RUN )
   END_RUNG
   RUNG wire#w1
      I_Contact( "IO Motor MCC Preparation_DB"."P-05.01".FB_ON )
      Coil( "T-21.00_DB".Tomato.P_STOP )
   END_RUNG
   // the same network as SCL:
   "T-21.00_DB".Tomato.ISTART_COND := NOT "T-20.00_DB".Tomato.QDOSERun AND NOT "T-30.00_DB".Tomato.QDOSERun AND NOT "T-31.00_DB".Tomato.QDOSERun AND "T-05.01_DB".State.Ready_For_Transfer;
   "T-21.00_DB".Tomato.V_OPEN := "T-21.00_DB".Tomato.ISTART_COND AND "IO_Valve_Blending_DB"."AV-21.12".FB_OPEN;
   "T-21.00_DB".Tomato.V_CLOSE := "T-21.00_DB".Tomato.ISTART_COND AND NOT "IO_Valve_Blending_DB"."AV-21.12".FB_OPEN;
   "T-21.00_DB".Tomato.P_RUN := "T-21.00_DB".Tomato.ISTART_COND AND "IO Motor MCC Preparation_DB"."P-05.01".FB_ON;
   "T-21.00_DB".Tomato.P_STOP := "T-21.00_DB".Tomato.ISTART_COND AND NOT "IO Motor MCC Preparation_DB"."P-05.01".FB_ON;
END_REGION

REGION Network 18: T-21_Dose_FreshChili_1
   RUNG wire#powerrail
      I_Contact( "T-20.00_DB".ChiliFresh_1.QDOSERun )
      I_Contact( "T-30.00_DB".ChiliFresh_1.QDOSERun )
      I_Contact( "T-31.00_DB".ChiliFresh_1.QDOSERun )
      Contact( "T-06.01_DB".State.Ready_For_Transfer )
      wire#w1
      Coil( "T-21.00_DB".ChiliFresh_1.ISTART_COND )
   END_RUNG
   RUNG wire#w1
      Contact( "IO_Valve_Blending_DB"."AV-21.05".FB_OPEN )
      Coil( "T-21.00_DB".ChiliFresh_1.V_OPEN )
   END_RUNG
   RUNG wire#w1
      I_Contact( "IO_Valve_Blending_DB"."AV-21.05".FB_OPEN )
      Coil( "T-21.00_DB".ChiliFresh_1.V_CLOSE )
   END_RUNG
   RUNG wire#w1
      Contact( "IO Motor MCC Preparation_DB"."P-06.01".FB_ON )
      Coil( "T-21.00_DB".ChiliFresh_1.P_RUN )
   END_RUNG
   RUNG wire#w1
      I_Contact( "IO Motor MCC Preparation_DB"."P-06.01".FB_ON )
      Coil( "T-21.00_DB".ChiliFresh_1.P_STOP )
   END_RUNG
   // the same network as SCL:
   "T-21.00_DB".ChiliFresh_1.ISTART_COND := NOT "T-20.00_DB".ChiliFresh_1.QDOSERun AND NOT "T-30.00_DB".ChiliFresh_1.QDOSERun AND NOT "T-31.00_DB".ChiliFresh_1.QDOSERun AND "T-06.01_DB".State.Ready_For_Transfer;
   "T-21.00_DB".ChiliFresh_1.V_OPEN := "T-21.00_DB".ChiliFresh_1.ISTART_COND AND "IO_Valve_Blending_DB"."AV-21.05".FB_OPEN;
   "T-21.00_DB".ChiliFresh_1.V_CLOSE := "T-21.00_DB".ChiliFresh_1.ISTART_COND AND NOT "IO_Valve_Blending_DB"."AV-21.05".FB_OPEN;
   "T-21.00_DB".ChiliFresh_1.P_RUN := "T-21.00_DB".ChiliFresh_1.ISTART_COND AND "IO Motor MCC Preparation_DB"."P-06.01".FB_ON;
   "T-21.00_DB".ChiliFresh_1.P_STOP := "T-21.00_DB".ChiliFresh_1.ISTART_COND AND NOT "IO Motor MCC Preparation_DB"."P-06.01".FB_ON;
END_REGION

REGION Network 19: T-21_Dose_FreshChili_2
   RUNG wire#powerrail
      I_Contact( "T-20.00_DB".ChiliFresh_2.QDOSERun )
      I_Contact( "T-30.00_DB".ChiliFresh_2.QDOSERun )
      I_Contact( "T-31.00_DB".ChiliFresh_2.QDOSERun )
      Contact( "T-07.01_DB".State.Ready_For_Transfer )
      wire#w1
      Coil( "T-21.00_DB".ChiliFresh_2.ISTART_COND )
   END_RUNG
   RUNG wire#w1
      Contact( "IO_Valve_Blending_DB"."AV-21.06".FB_OPEN )
      Coil( "T-21.00_DB".ChiliFresh_2.V_OPEN )
   END_RUNG
   RUNG wire#w1
      I_Contact( "IO_Valve_Blending_DB"."AV-21.06".FB_OPEN )
      Coil( "T-21.00_DB".ChiliFresh_2.V_CLOSE )
   END_RUNG
   RUNG wire#w1
      Contact( "IO Motor MCC Preparation_DB"."P-07.01".FB_ON )
      Coil( "T-21.00_DB".ChiliFresh_2.P_RUN )
   END_RUNG
   RUNG wire#w1
      I_Contact( "IO Motor MCC Preparation_DB"."P-07.01".FB_ON )
      Coil( "T-21.00_DB".ChiliFresh_2.P_STOP )
   END_RUNG
   // the same network as SCL:
   "T-21.00_DB".ChiliFresh_2.ISTART_COND := NOT "T-20.00_DB".ChiliFresh_2.QDOSERun AND NOT "T-30.00_DB".ChiliFresh_2.QDOSERun AND NOT "T-31.00_DB".ChiliFresh_2.QDOSERun AND "T-07.01_DB".State.Ready_For_Transfer;
   "T-21.00_DB".ChiliFresh_2.V_OPEN := "T-21.00_DB".ChiliFresh_2.ISTART_COND AND "IO_Valve_Blending_DB"."AV-21.06".FB_OPEN;
   "T-21.00_DB".ChiliFresh_2.V_CLOSE := "T-21.00_DB".ChiliFresh_2.ISTART_COND AND NOT "IO_Valve_Blending_DB"."AV-21.06".FB_OPEN;
   "T-21.00_DB".ChiliFresh_2.P_RUN := "T-21.00_DB".ChiliFresh_2.ISTART_COND AND "IO Motor MCC Preparation_DB"."P-07.01".FB_ON;
   "T-21.00_DB".ChiliFresh_2.P_STOP := "T-21.00_DB".ChiliFresh_2.ISTART_COND AND NOT "IO Motor MCC Preparation_DB"."P-07.01".FB_ON;
END_REGION

REGION Network 20: T-21_Dose_FreshChili_3
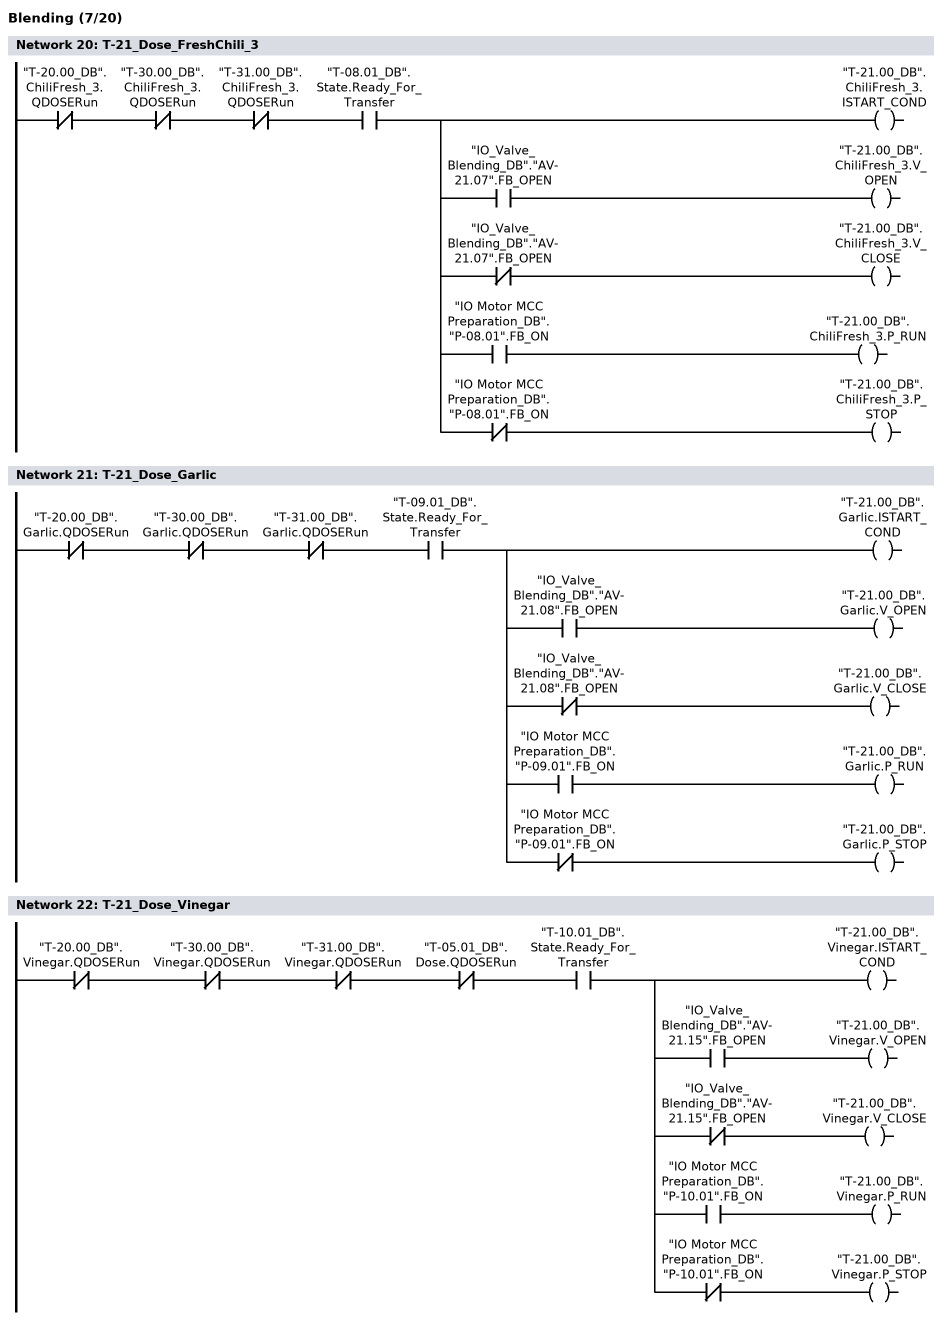
   RUNG wire#powerrail
      I_Contact( "T-20.00_DB".ChiliFresh_3.QDOSERun )
      I_Contact( "T-30.00_DB".ChiliFresh_3.QDOSERun )
      I_Contact( "T-31.00_DB".ChiliFresh_3.QDOSERun )
      Contact( "T-08.01_DB".State.Ready_For_Transfer )
      wire#w1
      Coil( "T-21.00_DB".ChiliFresh_3.ISTART_COND )
   END_RUNG
   RUNG wire#w1
      Contact( "IO_Valve_Blending_DB"."AV-21.07".FB_OPEN )
      Coil( "T-21.00_DB".ChiliFresh_3.V_OPEN )
   END_RUNG
   RUNG wire#w1
      I_Contact( "IO_Valve_Blending_DB"."AV-21.07".FB_OPEN )
      Coil( "T-21.00_DB".ChiliFresh_3.V_CLOSE )
   END_RUNG
   RUNG wire#w1
      Contact( "IO Motor MCC Preparation_DB"."P-08.01".FB_ON )
      Coil( "T-21.00_DB".ChiliFresh_3.P_RUN )
   END_RUNG
   RUNG wire#w1
      I_Contact( "IO Motor MCC Preparation_DB"."P-08.01".FB_ON )
      Coil( "T-21.00_DB".ChiliFresh_3.P_STOP )
   END_RUNG
   // the same network as SCL:
   "T-21.00_DB".ChiliFresh_3.ISTART_COND := NOT "T-20.00_DB".ChiliFresh_3.QDOSERun AND NOT "T-30.00_DB".ChiliFresh_3.QDOSERun AND NOT "T-31.00_DB".ChiliFresh_3.QDOSERun AND "T-08.01_DB".State.Ready_For_Transfer;
   "T-21.00_DB".ChiliFresh_3.V_OPEN := "T-21.00_DB".ChiliFresh_3.ISTART_COND AND "IO_Valve_Blending_DB"."AV-21.07".FB_OPEN;
   "T-21.00_DB".ChiliFresh_3.V_CLOSE := "T-21.00_DB".ChiliFresh_3.ISTART_COND AND NOT "IO_Valve_Blending_DB"."AV-21.07".FB_OPEN;
   "T-21.00_DB".ChiliFresh_3.P_RUN := "T-21.00_DB".ChiliFresh_3.ISTART_COND AND "IO Motor MCC Preparation_DB"."P-08.01".FB_ON;
   "T-21.00_DB".ChiliFresh_3.P_STOP := "T-21.00_DB".ChiliFresh_3.ISTART_COND AND NOT "IO Motor MCC Preparation_DB"."P-08.01".FB_ON;
END_REGION

REGION Network 21: T-21_Dose_Garlic
   RUNG wire#powerrail
      I_Contact( "T-20.00_DB".Garlic.QDOSERun )
      I_Contact( "T-30.00_DB".Garlic.QDOSERun )
      I_Contact( "T-31.00_DB".Garlic.QDOSERun )
      Contact( "T-09.01_DB".State.Ready_For_Transfer )
      wire#w1
      Coil( "T-21.00_DB".Garlic.ISTART_COND )
   END_RUNG
   RUNG wire#w1
      Contact( "IO_Valve_Blending_DB"."AV-21.08".FB_OPEN )
      Coil( "T-21.00_DB".Garlic.V_OPEN )
   END_RUNG
   RUNG wire#w1
      I_Contact( "IO_Valve_Blending_DB"."AV-21.08".FB_OPEN )
      Coil( "T-21.00_DB".Garlic.V_CLOSE )
   END_RUNG
   RUNG wire#w1
      Contact( "IO Motor MCC Preparation_DB"."P-09.01".FB_ON )
      Coil( "T-21.00_DB".Garlic.P_RUN )
   END_RUNG
   RUNG wire#w1
      I_Contact( "IO Motor MCC Preparation_DB"."P-09.01".FB_ON )
      Coil( "T-21.00_DB".Garlic.P_STOP )
   END_RUNG
   // the same network as SCL:
   "T-21.00_DB".Garlic.ISTART_COND := NOT "T-20.00_DB".Garlic.QDOSERun AND NOT "T-30.00_DB".Garlic.QDOSERun AND NOT "T-31.00_DB".Garlic.QDOSERun AND "T-09.01_DB".State.Ready_For_Transfer;
   "T-21.00_DB".Garlic.V_OPEN := "T-21.00_DB".Garlic.ISTART_COND AND "IO_Valve_Blending_DB"."AV-21.08".FB_OPEN;
   "T-21.00_DB".Garlic.V_CLOSE := "T-21.00_DB".Garlic.ISTART_COND AND NOT "IO_Valve_Blending_DB"."AV-21.08".FB_OPEN;
   "T-21.00_DB".Garlic.P_RUN := "T-21.00_DB".Garlic.ISTART_COND AND "IO Motor MCC Preparation_DB"."P-09.01".FB_ON;
   "T-21.00_DB".Garlic.P_STOP := "T-21.00_DB".Garlic.ISTART_COND AND NOT "IO Motor MCC Preparation_DB"."P-09.01".FB_ON;
END_REGION

REGION Network 22: T-21_Dose_Vinegar
   RUNG wire#powerrail
      I_Contact( "T-20.00_DB".Vinegar.QDOSERun )
      I_Contact( "T-30.00_DB".Vinegar.QDOSERun )
      I_Contact( "T-31.00_DB".Vinegar.QDOSERun )
      I_Contact( "T-05.01_DB".Dose.QDOSERun )
      Contact( "T-10.01_DB".State.Ready_For_Transfer )
      wire#w1
      Coil( "T-21.00_DB".Vinegar.ISTART_COND )
   END_RUNG
   RUNG wire#w1
      Contact( "IO_Valve_Blending_DB"."AV-21.15".FB_OPEN )
      Coil( "T-21.00_DB".Vinegar.V_OPEN )
   END_RUNG
   RUNG wire#w1
      I_Contact( "IO_Valve_Blending_DB"."AV-21.15".FB_OPEN )
      Coil( "T-21.00_DB".Vinegar.V_CLOSE )
   END_RUNG
   RUNG wire#w1
      Contact( "IO Motor MCC Preparation_DB"."P-10.01".FB_ON )
      Coil( "T-21.00_DB".Vinegar.P_RUN )
   END_RUNG
   RUNG wire#w1
      I_Contact( "IO Motor MCC Preparation_DB"."P-10.01".FB_ON )
      Coil( "T-21.00_DB".Vinegar.P_STOP )
   END_RUNG
   // the same network as SCL:
   "T-21.00_DB".Vinegar.ISTART_COND := NOT "T-20.00_DB".Vinegar.QDOSERun AND NOT "T-30.00_DB".Vinegar.QDOSERun AND NOT "T-31.00_DB".Vinegar.QDOSERun AND NOT "T-05.01_DB".Dose.QDOSERun AND "T-10.01_DB".State.Ready_For_Transfer;
   "T-21.00_DB".Vinegar.V_OPEN := "T-21.00_DB".Vinegar.ISTART_COND AND "IO_Valve_Blending_DB"."AV-21.15".FB_OPEN;
   "T-21.00_DB".Vinegar.V_CLOSE := "T-21.00_DB".Vinegar.ISTART_COND AND NOT "IO_Valve_Blending_DB"."AV-21.15".FB_OPEN;
   "T-21.00_DB".Vinegar.P_RUN := "T-21.00_DB".Vinegar.ISTART_COND AND "IO Motor MCC Preparation_DB"."P-10.01".FB_ON;
   "T-21.00_DB".Vinegar.P_STOP := "T-21.00_DB".Vinegar.ISTART_COND AND NOT "IO Motor MCC Preparation_DB"."P-10.01".FB_ON;
END_REGION

REGION Network 23: T-21.00
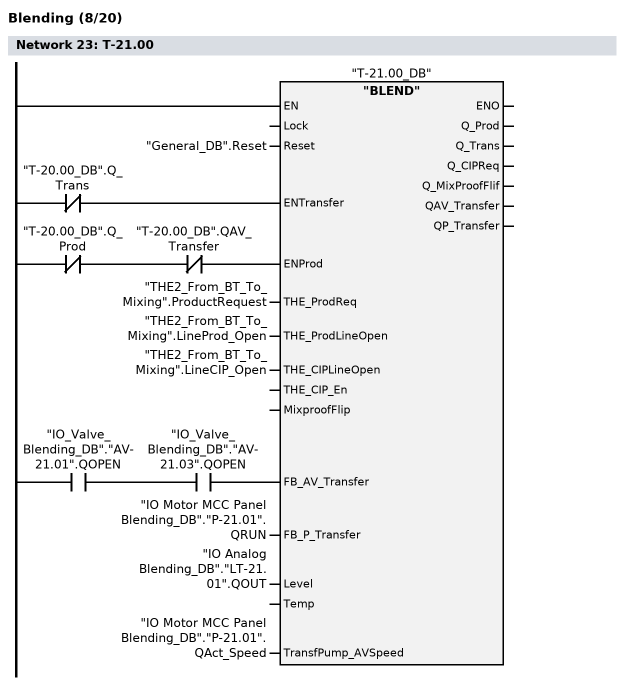
   RUNG wire#powerrail
      "T-21.00_DB"(ENTransfer := wire#w1, ENProd := wire#w2, FB_AV_Transfer := wire#w3, Lock :=, Reset := "General_DB".Reset, THE_ProdReq := "THE2_From_BT_To_Mixing".ProductRequest, THE_ProdLineOpen := "THE2_From_BT_To_Mixing".LineProd_Open, THE_CIPLineOpen := "THE2_From_BT_To_Mixing".LineCIP_Open, THE_CIP_En :=, MixproofFlip :=, FB_P_Transfer := "IO Motor MCC Panel Blending_DB"."P-21.01".QRUN, Level := "IO Analog Blending_DB"."LT-21.01".QOUT, Temp :=, TransfPump_AVSpeed := "IO Motor MCC Panel Blending_DB"."P-21.01".QAct_Speed, Q_Prod =>, Q_Trans =>, Q_CIPReq =>, Q_MixProofFlif =>, QAV_Transfer =>, QP_Transfer =>)
   END_RUNG
   RUNG wire#powerrail
      I_Contact( "T-20.00_DB".Q_Trans )
   END_RUNG wire#w1
   RUNG wire#powerrail
      I_Contact( "T-20.00_DB".Q_Prod )
      I_Contact( "T-20.00_DB".QAV_Transfer )
   END_RUNG wire#w2
   RUNG wire#powerrail
      Contact( "IO_Valve_Blending_DB"."AV-21.01".QOPEN )
      Contact( "IO_Valve_Blending_DB"."AV-21.03".QOPEN )
   END_RUNG wire#w3
   // the same network as SCL:
   "T-21.00_DB"(Reset := "General_DB".Reset,   // "BLEND"
                ENTransfer := NOT "T-20.00_DB".Q_Trans,
                ENProd := NOT "T-20.00_DB".Q_Prod AND NOT "T-20.00_DB".QAV_Transfer,
                THE_ProdReq := "THE2_From_BT_To_Mixing".ProductRequest,
                THE_ProdLineOpen := "THE2_From_BT_To_Mixing".LineProd_Open,
                THE_CIPLineOpen := "THE2_From_BT_To_Mixing".LineCIP_Open,
                FB_AV_Transfer := "IO_Valve_Blending_DB"."AV-21.01".QOPEN AND "IO_Valve_Blending_DB"."AV-21.03".QOPEN,
                FB_P_Transfer := "IO Motor MCC Panel Blending_DB"."P-21.01".QRUN,
                Level := "IO Analog Blending_DB"."LT-21.01".QOUT,
                TransfPump_AVSpeed := "IO Motor MCC Panel Blending_DB"."P-21.01".QAct_Speed);
END_REGION

REGION Network 24: Comm to Buffer Tank THE 2
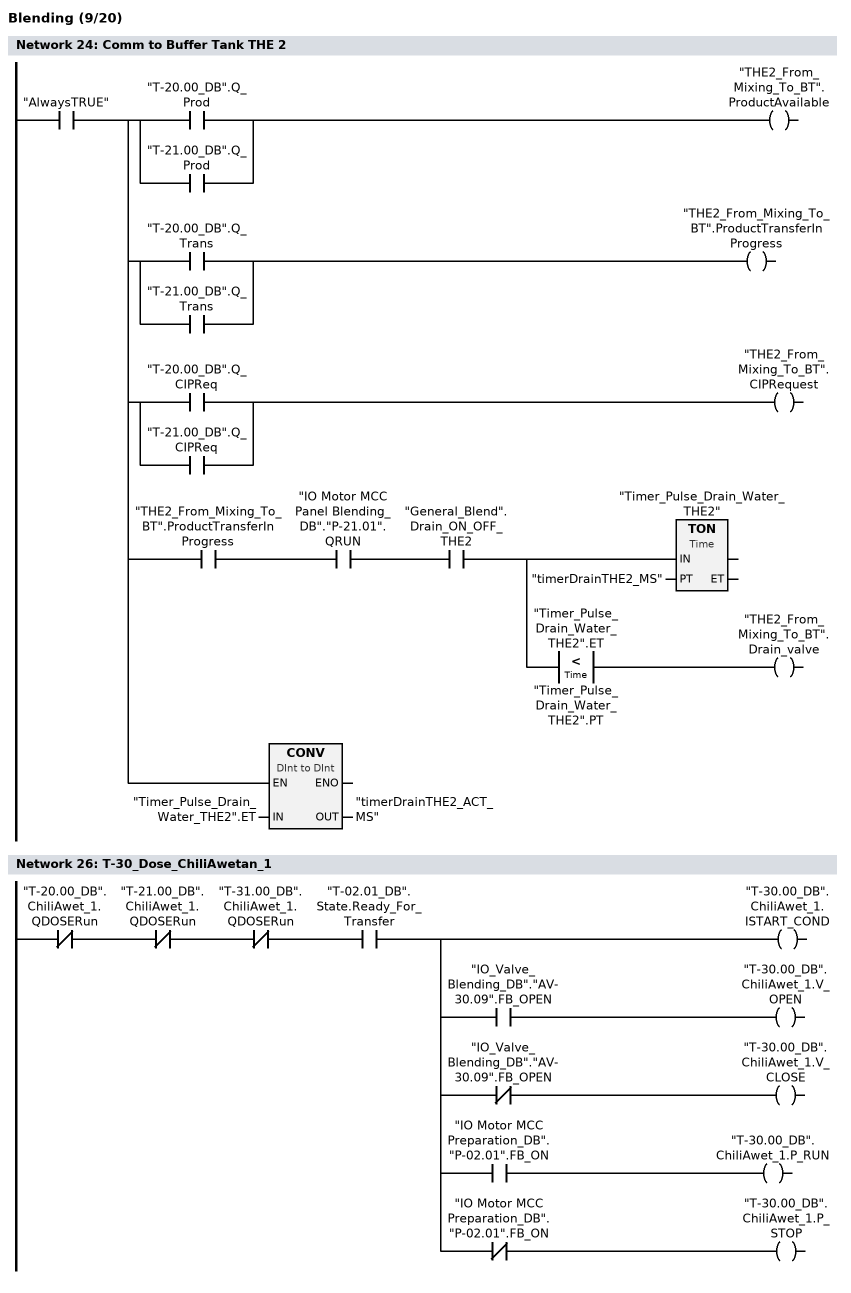
   RUNG wire#powerrail
      Contact( "AlwaysTRUE" )
      wire#w1
      Contact( "T-20.00_DB".Q_Prod )
      wire#w2
      Coil( "THE2_From_Mixing_To_BT".ProductAvailable )
   END_RUNG
   RUNG wire#w1
      Contact( "T-21.00_DB".Q_Prod )
   END_RUNG wire#w2
   RUNG wire#w1
      Contact( "T-20.00_DB".Q_Trans )
      wire#w3
      Coil( "THE2_From_Mixing_To_BT".ProductTransferInProgress )
   END_RUNG
   RUNG wire#w1
      Contact( "T-21.00_DB".Q_Trans )
   END_RUNG wire#w3
   RUNG wire#w1
      Contact( "T-20.00_DB".Q_CIPReq )
      wire#w4
      Coil( "THE2_From_Mixing_To_BT".CIPRequest )
   END_RUNG
   RUNG wire#w1
      Contact( "T-21.00_DB".Q_CIPReq )
   END_RUNG wire#w4
   RUNG wire#w1
      Contact( "THE2_From_Mixing_To_BT".ProductTransferInProgress )
      Contact( "IO Motor MCC Panel Blending_DB"."P-21.01".QRUN )
      Contact( "General_Blend".Drain_ON_OFF_THE2 )
      wire#w5
      { S7_Templates := "time_type := Time" } "Timer_Pulse_Drain_Water_THE2".TON(pt := "timerDrainTHE2_MS", et =>)
   END_RUNG
   RUNG wire#w5
      { S7_Templates := "SrcType := Time" } LT_Contact(in1 := "Timer_Pulse_Drain_Water_THE2".ET, in2 := "Timer_Pulse_Drain_Water_THE2".PT)
      Coil( "THE2_From_Mixing_To_BT".Drain_valve )
   END_RUNG
   RUNG wire#w1
      { S7_Templates := "[SrcType := DInt, DestType := DInt]" } Convert(in := "Timer_Pulse_Drain_Water_THE2".ET, out => "timerDrainTHE2_ACT_MS")
   END_RUNG
   // the same network as SCL:
   "THE2_From_Mixing_To_BT".ProductAvailable := "AlwaysTRUE" AND ("T-20.00_DB".Q_Prod OR "T-21.00_DB".Q_Prod);
   "THE2_From_Mixing_To_BT".ProductTransferInProgress := "AlwaysTRUE" AND ("T-20.00_DB".Q_Trans OR "T-21.00_DB".Q_Trans);
   "THE2_From_Mixing_To_BT".CIPRequest := "AlwaysTRUE" AND ("T-20.00_DB".Q_CIPReq OR "T-21.00_DB".Q_CIPReq);
   #_w1 := "AlwaysTRUE" AND "THE2_From_Mixing_To_BT".ProductTransferInProgress AND "IO Motor MCC Panel Blending_DB"."P-21.01".QRUN AND "General_Blend".Drain_ON_OFF_THE2;
   "Timer_Pulse_Drain_Water_THE2".TON(IN := #_w1, PT := "timerDrainTHE2_MS");
   "THE2_From_Mixing_To_BT".Drain_valve := #_w1 AND ("Timer_Pulse_Drain_Water_THE2".ET < "Timer_Pulse_Drain_Water_THE2".PT);
   IF "AlwaysTRUE" THEN "timerDrainTHE2_ACT_MS" := DINT_TO_DINT("Timer_Pulse_Drain_Water_THE2".ET); END_IF;
END_REGION

REGION Network 26: T-30_Dose_ChiliAwetan_1
   RUNG wire#powerrail
      I_Contact( "T-20.00_DB".ChiliAwet_1.QDOSERun )
      I_Contact( "T-21.00_DB".ChiliAwet_1.QDOSERun )
      I_Contact( "T-31.00_DB".ChiliAwet_1.QDOSERun )
      Contact( "T-02.01_DB".State.Ready_For_Transfer )
      wire#w1
      Coil( "T-30.00_DB".ChiliAwet_1.ISTART_COND )
   END_RUNG
   RUNG wire#w1
      Contact( "IO_Valve_Blending_DB"."AV-30.09".FB_OPEN )
      Coil( "T-30.00_DB".ChiliAwet_1.V_OPEN )
   END_RUNG
   RUNG wire#w1
      I_Contact( "IO_Valve_Blending_DB"."AV-30.09".FB_OPEN )
      Coil( "T-30.00_DB".ChiliAwet_1.V_CLOSE )
   END_RUNG
   RUNG wire#w1
      Contact( "IO Motor MCC Preparation_DB"."P-02.01".FB_ON )
      Coil( "T-30.00_DB".ChiliAwet_1.P_RUN )
   END_RUNG
   RUNG wire#w1
      I_Contact( "IO Motor MCC Preparation_DB"."P-02.01".FB_ON )
      Coil( "T-30.00_DB".ChiliAwet_1.P_STOP )
   END_RUNG
   // the same network as SCL:
   "T-30.00_DB".ChiliAwet_1.ISTART_COND := NOT "T-20.00_DB".ChiliAwet_1.QDOSERun AND NOT "T-21.00_DB".ChiliAwet_1.QDOSERun AND NOT "T-31.00_DB".ChiliAwet_1.QDOSERun AND "T-02.01_DB".State.Ready_For_Transfer;
   "T-30.00_DB".ChiliAwet_1.V_OPEN := "T-30.00_DB".ChiliAwet_1.ISTART_COND AND "IO_Valve_Blending_DB"."AV-30.09".FB_OPEN;
   "T-30.00_DB".ChiliAwet_1.V_CLOSE := "T-30.00_DB".ChiliAwet_1.ISTART_COND AND NOT "IO_Valve_Blending_DB"."AV-30.09".FB_OPEN;
   "T-30.00_DB".ChiliAwet_1.P_RUN := "T-30.00_DB".ChiliAwet_1.ISTART_COND AND "IO Motor MCC Preparation_DB"."P-02.01".FB_ON;
   "T-30.00_DB".ChiliAwet_1.P_STOP := "T-30.00_DB".ChiliAwet_1.ISTART_COND AND NOT "IO Motor MCC Preparation_DB"."P-02.01".FB_ON;
END_REGION

REGION Network 27: T-30_Dose_ChiliAwetan_2
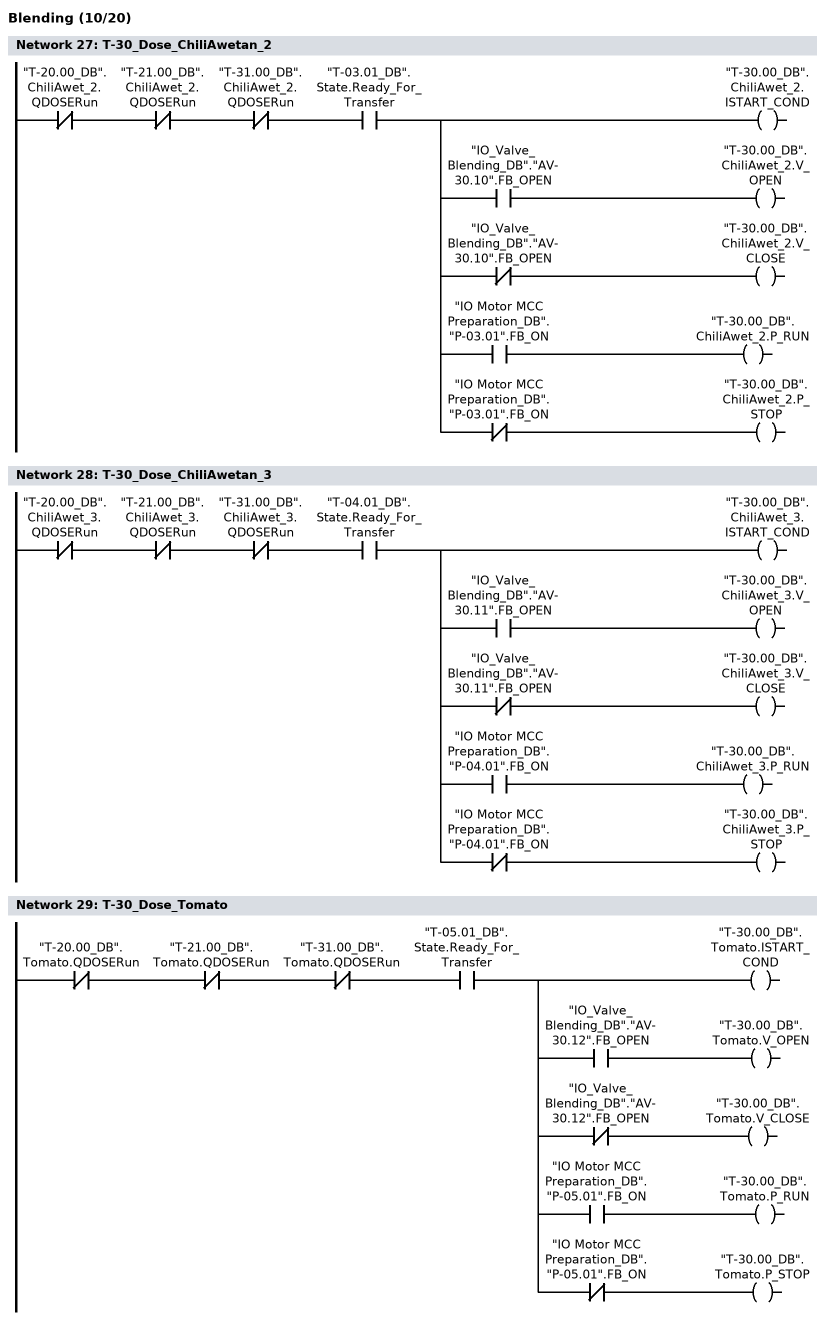
   RUNG wire#powerrail
      I_Contact( "T-20.00_DB".ChiliAwet_2.QDOSERun )
      I_Contact( "T-21.00_DB".ChiliAwet_2.QDOSERun )
      I_Contact( "T-31.00_DB".ChiliAwet_2.QDOSERun )
      Contact( "T-03.01_DB".State.Ready_For_Transfer )
      wire#w1
      Coil( "T-30.00_DB".ChiliAwet_2.ISTART_COND )
   END_RUNG
   RUNG wire#w1
      Contact( "IO_Valve_Blending_DB"."AV-30.10".FB_OPEN )
      Coil( "T-30.00_DB".ChiliAwet_2.V_OPEN )
   END_RUNG
   RUNG wire#w1
      I_Contact( "IO_Valve_Blending_DB"."AV-30.10".FB_OPEN )
      Coil( "T-30.00_DB".ChiliAwet_2.V_CLOSE )
   END_RUNG
   RUNG wire#w1
      Contact( "IO Motor MCC Preparation_DB"."P-03.01".FB_ON )
      Coil( "T-30.00_DB".ChiliAwet_2.P_RUN )
   END_RUNG
   RUNG wire#w1
      I_Contact( "IO Motor MCC Preparation_DB"."P-03.01".FB_ON )
      Coil( "T-30.00_DB".ChiliAwet_2.P_STOP )
   END_RUNG
   // the same network as SCL:
   "T-30.00_DB".ChiliAwet_2.ISTART_COND := NOT "T-20.00_DB".ChiliAwet_2.QDOSERun AND NOT "T-21.00_DB".ChiliAwet_2.QDOSERun AND NOT "T-31.00_DB".ChiliAwet_2.QDOSERun AND "T-03.01_DB".State.Ready_For_Transfer;
   "T-30.00_DB".ChiliAwet_2.V_OPEN := "T-30.00_DB".ChiliAwet_2.ISTART_COND AND "IO_Valve_Blending_DB"."AV-30.10".FB_OPEN;
   "T-30.00_DB".ChiliAwet_2.V_CLOSE := "T-30.00_DB".ChiliAwet_2.ISTART_COND AND NOT "IO_Valve_Blending_DB"."AV-30.10".FB_OPEN;
   "T-30.00_DB".ChiliAwet_2.P_RUN := "T-30.00_DB".ChiliAwet_2.ISTART_COND AND "IO Motor MCC Preparation_DB"."P-03.01".FB_ON;
   "T-30.00_DB".ChiliAwet_2.P_STOP := "T-30.00_DB".ChiliAwet_2.ISTART_COND AND NOT "IO Motor MCC Preparation_DB"."P-03.01".FB_ON;
END_REGION

REGION Network 28: T-30_Dose_ChiliAwetan_3
   RUNG wire#powerrail
      I_Contact( "T-20.00_DB".ChiliAwet_3.QDOSERun )
      I_Contact( "T-21.00_DB".ChiliAwet_3.QDOSERun )
      I_Contact( "T-31.00_DB".ChiliAwet_3.QDOSERun )
      Contact( "T-04.01_DB".State.Ready_For_Transfer )
      wire#w1
      Coil( "T-30.00_DB".ChiliAwet_3.ISTART_COND )
   END_RUNG
   RUNG wire#w1
      Contact( "IO_Valve_Blending_DB"."AV-30.11".FB_OPEN )
      Coil( "T-30.00_DB".ChiliAwet_3.V_OPEN )
   END_RUNG
   RUNG wire#w1
      I_Contact( "IO_Valve_Blending_DB"."AV-30.11".FB_OPEN )
      Coil( "T-30.00_DB".ChiliAwet_3.V_CLOSE )
   END_RUNG
   RUNG wire#w1
      Contact( "IO Motor MCC Preparation_DB"."P-04.01".FB_ON )
      Coil( "T-30.00_DB".ChiliAwet_3.P_RUN )
   END_RUNG
   RUNG wire#w1
      I_Contact( "IO Motor MCC Preparation_DB"."P-04.01".FB_ON )
      Coil( "T-30.00_DB".ChiliAwet_3.P_STOP )
   END_RUNG
   // the same network as SCL:
   "T-30.00_DB".ChiliAwet_3.ISTART_COND := NOT "T-20.00_DB".ChiliAwet_3.QDOSERun AND NOT "T-21.00_DB".ChiliAwet_3.QDOSERun AND NOT "T-31.00_DB".ChiliAwet_3.QDOSERun AND "T-04.01_DB".State.Ready_For_Transfer;
   "T-30.00_DB".ChiliAwet_3.V_OPEN := "T-30.00_DB".ChiliAwet_3.ISTART_COND AND "IO_Valve_Blending_DB"."AV-30.11".FB_OPEN;
   "T-30.00_DB".ChiliAwet_3.V_CLOSE := "T-30.00_DB".ChiliAwet_3.ISTART_COND AND NOT "IO_Valve_Blending_DB"."AV-30.11".FB_OPEN;
   "T-30.00_DB".ChiliAwet_3.P_RUN := "T-30.00_DB".ChiliAwet_3.ISTART_COND AND "IO Motor MCC Preparation_DB"."P-04.01".FB_ON;
   "T-30.00_DB".ChiliAwet_3.P_STOP := "T-30.00_DB".ChiliAwet_3.ISTART_COND AND NOT "IO Motor MCC Preparation_DB"."P-04.01".FB_ON;
END_REGION

REGION Network 29: T-30_Dose_Tomato
   RUNG wire#powerrail
      I_Contact( "T-20.00_DB".Tomato.QDOSERun )
      I_Contact( "T-21.00_DB".Tomato.QDOSERun )
      I_Contact( "T-31.00_DB".Tomato.QDOSERun )
      Contact( "T-05.01_DB".State.Ready_For_Transfer )
      wire#w1
      Coil( "T-30.00_DB".Tomato.ISTART_COND )
   END_RUNG
   RUNG wire#w1
      Contact( "IO_Valve_Blending_DB"."AV-30.12".FB_OPEN )
      Coil( "T-30.00_DB".Tomato.V_OPEN )
   END_RUNG
   RUNG wire#w1
      I_Contact( "IO_Valve_Blending_DB"."AV-30.12".FB_OPEN )
      Coil( "T-30.00_DB".Tomato.V_CLOSE )
   END_RUNG
   RUNG wire#w1
      Contact( "IO Motor MCC Preparation_DB"."P-05.01".FB_ON )
      Coil( "T-30.00_DB".Tomato.P_RUN )
   END_RUNG
   RUNG wire#w1
      I_Contact( "IO Motor MCC Preparation_DB"."P-05.01".FB_ON )
      Coil( "T-30.00_DB".Tomato.P_STOP )
   END_RUNG
   // the same network as SCL:
   "T-30.00_DB".Tomato.ISTART_COND := NOT "T-20.00_DB".Tomato.QDOSERun AND NOT "T-21.00_DB".Tomato.QDOSERun AND NOT "T-31.00_DB".Tomato.QDOSERun AND "T-05.01_DB".State.Ready_For_Transfer;
   "T-30.00_DB".Tomato.V_OPEN := "T-30.00_DB".Tomato.ISTART_COND AND "IO_Valve_Blending_DB"."AV-30.12".FB_OPEN;
   "T-30.00_DB".Tomato.V_CLOSE := "T-30.00_DB".Tomato.ISTART_COND AND NOT "IO_Valve_Blending_DB"."AV-30.12".FB_OPEN;
   "T-30.00_DB".Tomato.P_RUN := "T-30.00_DB".Tomato.ISTART_COND AND "IO Motor MCC Preparation_DB"."P-05.01".FB_ON;
   "T-30.00_DB".Tomato.P_STOP := "T-30.00_DB".Tomato.ISTART_COND AND NOT "IO Motor MCC Preparation_DB"."P-05.01".FB_ON;
END_REGION

REGION Network 30: T-30_Dose_FreshChili_1
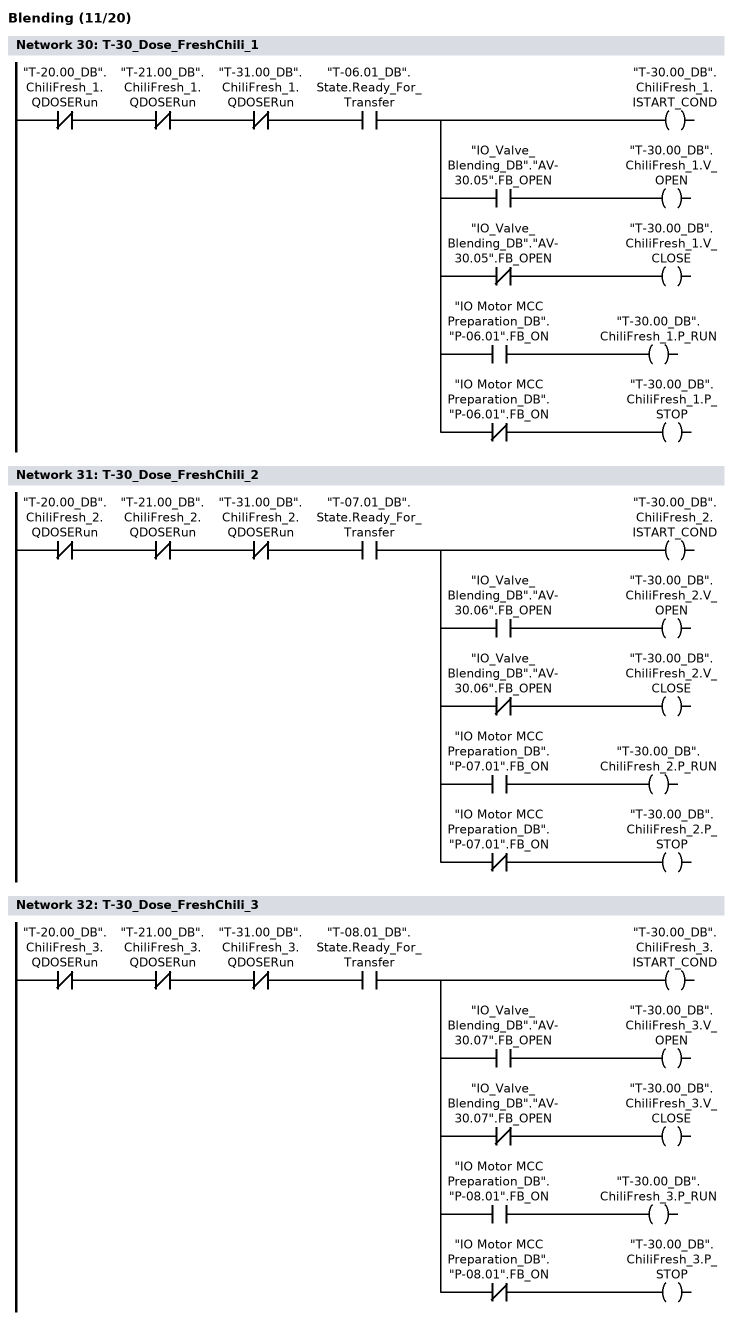
   RUNG wire#powerrail
      I_Contact( "T-20.00_DB".ChiliFresh_1.QDOSERun )
      I_Contact( "T-21.00_DB".ChiliFresh_1.QDOSERun )
      I_Contact( "T-31.00_DB".ChiliFresh_1.QDOSERun )
      Contact( "T-06.01_DB".State.Ready_For_Transfer )
      wire#w1
      Coil( "T-30.00_DB".ChiliFresh_1.ISTART_COND )
   END_RUNG
   RUNG wire#w1
      Contact( "IO_Valve_Blending_DB"."AV-30.05".FB_OPEN )
      Coil( "T-30.00_DB".ChiliFresh_1.V_OPEN )
   END_RUNG
   RUNG wire#w1
      I_Contact( "IO_Valve_Blending_DB"."AV-30.05".FB_OPEN )
      Coil( "T-30.00_DB".ChiliFresh_1.V_CLOSE )
   END_RUNG
   RUNG wire#w1
      Contact( "IO Motor MCC Preparation_DB"."P-06.01".FB_ON )
      Coil( "T-30.00_DB".ChiliFresh_1.P_RUN )
   END_RUNG
   RUNG wire#w1
      I_Contact( "IO Motor MCC Preparation_DB"."P-06.01".FB_ON )
      Coil( "T-30.00_DB".ChiliFresh_1.P_STOP )
   END_RUNG
   // the same network as SCL:
   "T-30.00_DB".ChiliFresh_1.ISTART_COND := NOT "T-20.00_DB".ChiliFresh_1.QDOSERun AND NOT "T-21.00_DB".ChiliFresh_1.QDOSERun AND NOT "T-31.00_DB".ChiliFresh_1.QDOSERun AND "T-06.01_DB".State.Ready_For_Transfer;
   "T-30.00_DB".ChiliFresh_1.V_OPEN := "T-30.00_DB".ChiliFresh_1.ISTART_COND AND "IO_Valve_Blending_DB"."AV-30.05".FB_OPEN;
   "T-30.00_DB".ChiliFresh_1.V_CLOSE := "T-30.00_DB".ChiliFresh_1.ISTART_COND AND NOT "IO_Valve_Blending_DB"."AV-30.05".FB_OPEN;
   "T-30.00_DB".ChiliFresh_1.P_RUN := "T-30.00_DB".ChiliFresh_1.ISTART_COND AND "IO Motor MCC Preparation_DB"."P-06.01".FB_ON;
   "T-30.00_DB".ChiliFresh_1.P_STOP := "T-30.00_DB".ChiliFresh_1.ISTART_COND AND NOT "IO Motor MCC Preparation_DB"."P-06.01".FB_ON;
END_REGION

REGION Network 31: T-30_Dose_FreshChili_2
   RUNG wire#powerrail
      I_Contact( "T-20.00_DB".ChiliFresh_2.QDOSERun )
      I_Contact( "T-21.00_DB".ChiliFresh_2.QDOSERun )
      I_Contact( "T-31.00_DB".ChiliFresh_2.QDOSERun )
      Contact( "T-07.01_DB".State.Ready_For_Transfer )
      wire#w1
      Coil( "T-30.00_DB".ChiliFresh_2.ISTART_COND )
   END_RUNG
   RUNG wire#w1
      Contact( "IO_Valve_Blending_DB"."AV-30.06".FB_OPEN )
      Coil( "T-30.00_DB".ChiliFresh_2.V_OPEN )
   END_RUNG
   RUNG wire#w1
      I_Contact( "IO_Valve_Blending_DB"."AV-30.06".FB_OPEN )
      Coil( "T-30.00_DB".ChiliFresh_2.V_CLOSE )
   END_RUNG
   RUNG wire#w1
      Contact( "IO Motor MCC Preparation_DB"."P-07.01".FB_ON )
      Coil( "T-30.00_DB".ChiliFresh_2.P_RUN )
   END_RUNG
   RUNG wire#w1
      I_Contact( "IO Motor MCC Preparation_DB"."P-07.01".FB_ON )
      Coil( "T-30.00_DB".ChiliFresh_2.P_STOP )
   END_RUNG
   // the same network as SCL:
   "T-30.00_DB".ChiliFresh_2.ISTART_COND := NOT "T-20.00_DB".ChiliFresh_2.QDOSERun AND NOT "T-21.00_DB".ChiliFresh_2.QDOSERun AND NOT "T-31.00_DB".ChiliFresh_2.QDOSERun AND "T-07.01_DB".State.Ready_For_Transfer;
   "T-30.00_DB".ChiliFresh_2.V_OPEN := "T-30.00_DB".ChiliFresh_2.ISTART_COND AND "IO_Valve_Blending_DB"."AV-30.06".FB_OPEN;
   "T-30.00_DB".ChiliFresh_2.V_CLOSE := "T-30.00_DB".ChiliFresh_2.ISTART_COND AND NOT "IO_Valve_Blending_DB"."AV-30.06".FB_OPEN;
   "T-30.00_DB".ChiliFresh_2.P_RUN := "T-30.00_DB".ChiliFresh_2.ISTART_COND AND "IO Motor MCC Preparation_DB"."P-07.01".FB_ON;
   "T-30.00_DB".ChiliFresh_2.P_STOP := "T-30.00_DB".ChiliFresh_2.ISTART_COND AND NOT "IO Motor MCC Preparation_DB"."P-07.01".FB_ON;
END_REGION

REGION Network 32: T-30_Dose_FreshChili_3
   RUNG wire#powerrail
      I_Contact( "T-20.00_DB".ChiliFresh_3.QDOSERun )
      I_Contact( "T-21.00_DB".ChiliFresh_3.QDOSERun )
      I_Contact( "T-31.00_DB".ChiliFresh_3.QDOSERun )
      Contact( "T-08.01_DB".State.Ready_For_Transfer )
      wire#w1
      Coil( "T-30.00_DB".ChiliFresh_3.ISTART_COND )
   END_RUNG
   RUNG wire#w1
      Contact( "IO_Valve_Blending_DB"."AV-30.07".FB_OPEN )
      Coil( "T-30.00_DB".ChiliFresh_3.V_OPEN )
   END_RUNG
   RUNG wire#w1
      I_Contact( "IO_Valve_Blending_DB"."AV-30.07".FB_OPEN )
      Coil( "T-30.00_DB".ChiliFresh_3.V_CLOSE )
   END_RUNG
   RUNG wire#w1
      Contact( "IO Motor MCC Preparation_DB"."P-08.01".FB_ON )
      Coil( "T-30.00_DB".ChiliFresh_3.P_RUN )
   END_RUNG
   RUNG wire#w1
      I_Contact( "IO Motor MCC Preparation_DB"."P-08.01".FB_ON )
      Coil( "T-30.00_DB".ChiliFresh_3.P_STOP )
   END_RUNG
   // the same network as SCL:
   "T-30.00_DB".ChiliFresh_3.ISTART_COND := NOT "T-20.00_DB".ChiliFresh_3.QDOSERun AND NOT "T-21.00_DB".ChiliFresh_3.QDOSERun AND NOT "T-31.00_DB".ChiliFresh_3.QDOSERun AND "T-08.01_DB".State.Ready_For_Transfer;
   "T-30.00_DB".ChiliFresh_3.V_OPEN := "T-30.00_DB".ChiliFresh_3.ISTART_COND AND "IO_Valve_Blending_DB"."AV-30.07".FB_OPEN;
   "T-30.00_DB".ChiliFresh_3.V_CLOSE := "T-30.00_DB".ChiliFresh_3.ISTART_COND AND NOT "IO_Valve_Blending_DB"."AV-30.07".FB_OPEN;
   "T-30.00_DB".ChiliFresh_3.P_RUN := "T-30.00_DB".ChiliFresh_3.ISTART_COND AND "IO Motor MCC Preparation_DB"."P-08.01".FB_ON;
   "T-30.00_DB".ChiliFresh_3.P_STOP := "T-30.00_DB".ChiliFresh_3.ISTART_COND AND NOT "IO Motor MCC Preparation_DB"."P-08.01".FB_ON;
END_REGION

REGION Network 33: T-30_Dose_Garlic
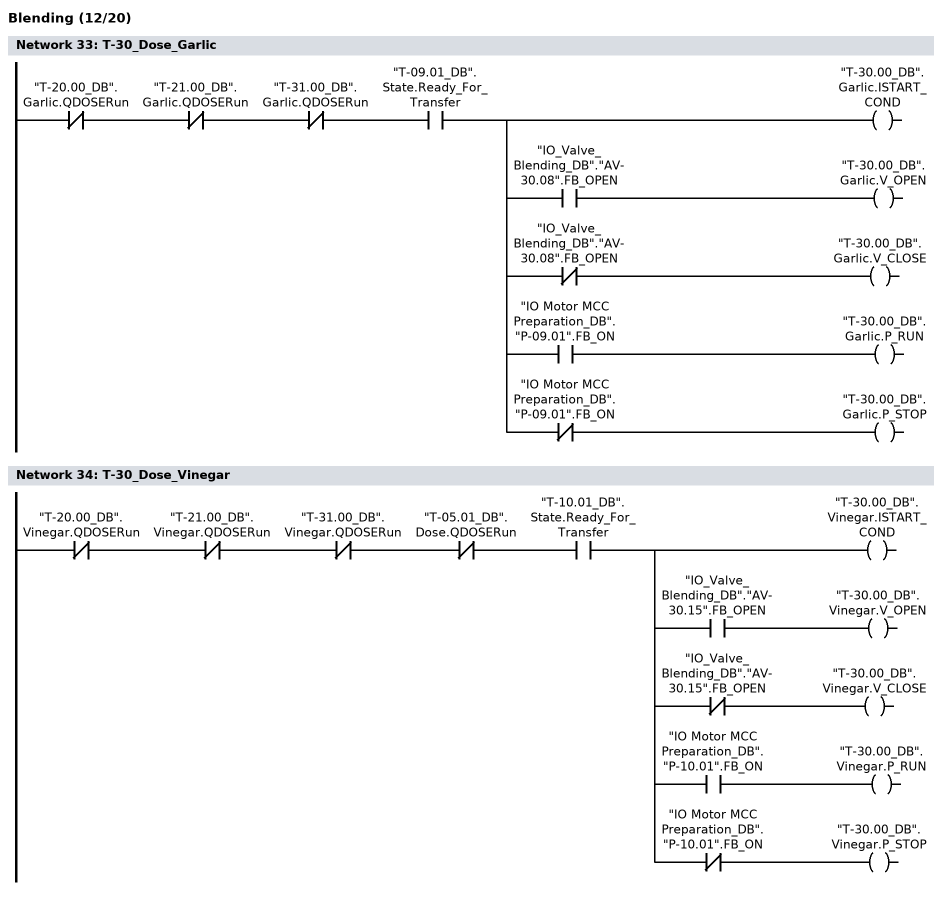
   RUNG wire#powerrail
      I_Contact( "T-20.00_DB".Garlic.QDOSERun )
      I_Contact( "T-21.00_DB".Garlic.QDOSERun )
      I_Contact( "T-31.00_DB".Garlic.QDOSERun )
      Contact( "T-09.01_DB".State.Ready_For_Transfer )
      wire#w1
      Coil( "T-30.00_DB".Garlic.ISTART_COND )
   END_RUNG
   RUNG wire#w1
      Contact( "IO_Valve_Blending_DB"."AV-30.08".FB_OPEN )
      Coil( "T-30.00_DB".Garlic.V_OPEN )
   END_RUNG
   RUNG wire#w1
      I_Contact( "IO_Valve_Blending_DB"."AV-30.08".FB_OPEN )
      Coil( "T-30.00_DB".Garlic.V_CLOSE )
   END_RUNG
   RUNG wire#w1
      Contact( "IO Motor MCC Preparation_DB"."P-09.01".FB_ON )
      Coil( "T-30.00_DB".Garlic.P_RUN )
   END_RUNG
   RUNG wire#w1
      I_Contact( "IO Motor MCC Preparation_DB"."P-09.01".FB_ON )
      Coil( "T-30.00_DB".Garlic.P_STOP )
   END_RUNG
   // the same network as SCL:
   "T-30.00_DB".Garlic.ISTART_COND := NOT "T-20.00_DB".Garlic.QDOSERun AND NOT "T-21.00_DB".Garlic.QDOSERun AND NOT "T-31.00_DB".Garlic.QDOSERun AND "T-09.01_DB".State.Ready_For_Transfer;
   "T-30.00_DB".Garlic.V_OPEN := "T-30.00_DB".Garlic.ISTART_COND AND "IO_Valve_Blending_DB"."AV-30.08".FB_OPEN;
   "T-30.00_DB".Garlic.V_CLOSE := "T-30.00_DB".Garlic.ISTART_COND AND NOT "IO_Valve_Blending_DB"."AV-30.08".FB_OPEN;
   "T-30.00_DB".Garlic.P_RUN := "T-30.00_DB".Garlic.ISTART_COND AND "IO Motor MCC Preparation_DB"."P-09.01".FB_ON;
   "T-30.00_DB".Garlic.P_STOP := "T-30.00_DB".Garlic.ISTART_COND AND NOT "IO Motor MCC Preparation_DB"."P-09.01".FB_ON;
END_REGION

REGION Network 34: T-30_Dose_Vinegar
   RUNG wire#powerrail
      I_Contact( "T-20.00_DB".Vinegar.QDOSERun )
      I_Contact( "T-21.00_DB".Vinegar.QDOSERun )
      I_Contact( "T-31.00_DB".Vinegar.QDOSERun )
      I_Contact( "T-05.01_DB".Dose.QDOSERun )
      Contact( "T-10.01_DB".State.Ready_For_Transfer )
      wire#w1
      Coil( "T-30.00_DB".Vinegar.ISTART_COND )
   END_RUNG
   RUNG wire#w1
      Contact( "IO_Valve_Blending_DB"."AV-30.15".FB_OPEN )
      Coil( "T-30.00_DB".Vinegar.V_OPEN )
   END_RUNG
   RUNG wire#w1
      I_Contact( "IO_Valve_Blending_DB"."AV-30.15".FB_OPEN )
      Coil( "T-30.00_DB".Vinegar.V_CLOSE )
   END_RUNG
   RUNG wire#w1
      Contact( "IO Motor MCC Preparation_DB"."P-10.01".FB_ON )
      Coil( "T-30.00_DB".Vinegar.P_RUN )
   END_RUNG
   RUNG wire#w1
      I_Contact( "IO Motor MCC Preparation_DB"."P-10.01".FB_ON )
      Coil( "T-30.00_DB".Vinegar.P_STOP )
   END_RUNG
   // the same network as SCL:
   "T-30.00_DB".Vinegar.ISTART_COND := NOT "T-20.00_DB".Vinegar.QDOSERun AND NOT "T-21.00_DB".Vinegar.QDOSERun AND NOT "T-31.00_DB".Vinegar.QDOSERun AND NOT "T-05.01_DB".Dose.QDOSERun AND "T-10.01_DB".State.Ready_For_Transfer;
   "T-30.00_DB".Vinegar.V_OPEN := "T-30.00_DB".Vinegar.ISTART_COND AND "IO_Valve_Blending_DB"."AV-30.15".FB_OPEN;
   "T-30.00_DB".Vinegar.V_CLOSE := "T-30.00_DB".Vinegar.ISTART_COND AND NOT "IO_Valve_Blending_DB"."AV-30.15".FB_OPEN;
   "T-30.00_DB".Vinegar.P_RUN := "T-30.00_DB".Vinegar.ISTART_COND AND "IO Motor MCC Preparation_DB"."P-10.01".FB_ON;
   "T-30.00_DB".Vinegar.P_STOP := "T-30.00_DB".Vinegar.ISTART_COND AND NOT "IO Motor MCC Preparation_DB"."P-10.01".FB_ON;
END_REGION

REGION Network 35: T-30.00
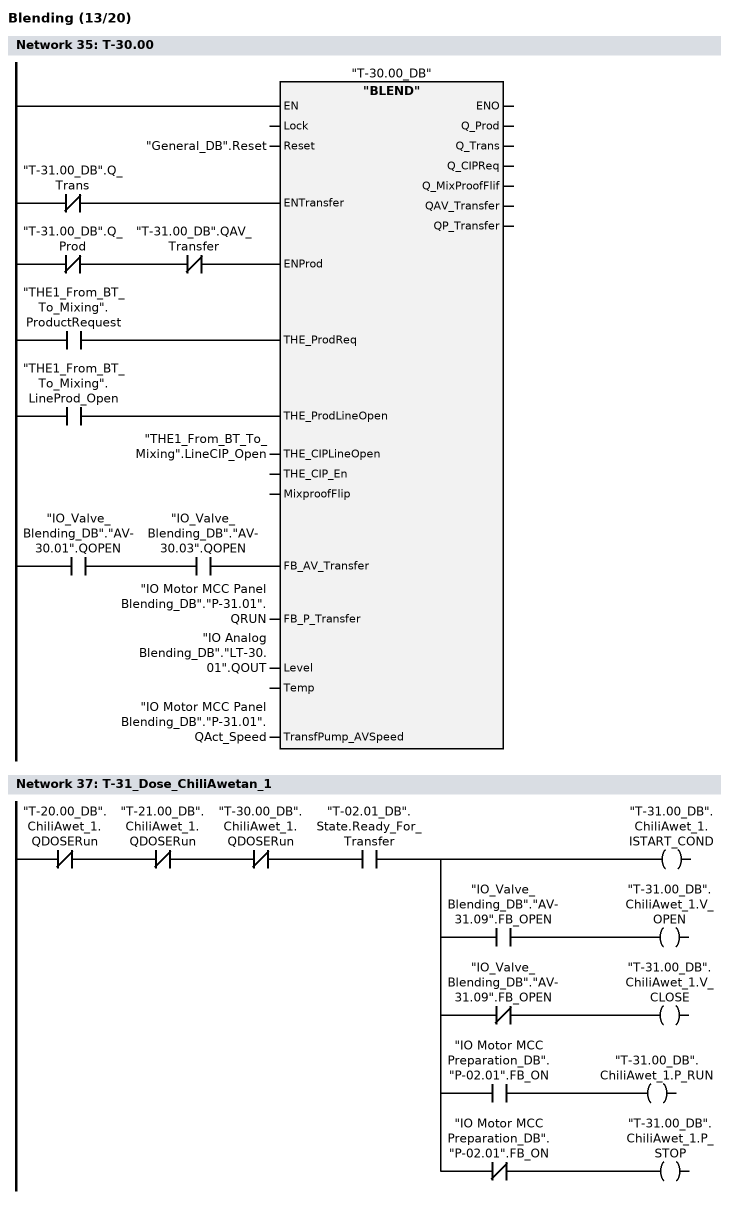
   RUNG wire#powerrail
      "T-30.00_DB"(ENTransfer := wire#w1, ENProd := wire#w2, THE_ProdReq := wire#w3, THE_ProdLineOpen := wire#w4, FB_AV_Transfer := wire#w5, Lock :=, Reset := "General_DB".Reset, THE_CIPLineOpen := "THE1_From_BT_To_Mixing".LineCIP_Open, THE_CIP_En :=, MixproofFlip :=, FB_P_Transfer := "IO Motor MCC Panel Blending_DB"."P-31.01".QRUN, Level := "IO Analog Blending_DB"."LT-30.01".QOUT, Temp :=, TransfPump_AVSpeed := "IO Motor MCC Panel Blending_DB"."P-31.01".QAct_Speed, Q_Prod =>, Q_Trans =>, Q_CIPReq =>, Q_MixProofFlif =>, QAV_Transfer =>, QP_Transfer =>)
   END_RUNG
   RUNG wire#powerrail
      I_Contact( "T-31.00_DB".Q_Trans )
   END_RUNG wire#w1
   RUNG wire#powerrail
      I_Contact( "T-31.00_DB".Q_Prod )
      I_Contact( "T-31.00_DB".QAV_Transfer )
   END_RUNG wire#w2
   RUNG wire#powerrail
      Contact( "THE1_From_BT_To_Mixing".ProductRequest )
   END_RUNG wire#w3
   RUNG wire#powerrail
      Contact( "THE1_From_BT_To_Mixing".LineProd_Open )
   END_RUNG wire#w4
   RUNG wire#powerrail
      Contact( "IO_Valve_Blending_DB"."AV-30.01".QOPEN )
      Contact( "IO_Valve_Blending_DB"."AV-30.03".QOPEN )
   END_RUNG wire#w5
   // the same network as SCL:
   "T-30.00_DB"(Reset := "General_DB".Reset,   // "BLEND"
                ENTransfer := NOT "T-31.00_DB".Q_Trans,
                ENProd := NOT "T-31.00_DB".Q_Prod AND NOT "T-31.00_DB".QAV_Transfer,
                THE_ProdReq := "THE1_From_BT_To_Mixing".ProductRequest,
                THE_ProdLineOpen := "THE1_From_BT_To_Mixing".LineProd_Open,
                THE_CIPLineOpen := "THE1_From_BT_To_Mixing".LineCIP_Open,
                FB_AV_Transfer := "IO_Valve_Blending_DB"."AV-30.01".QOPEN AND "IO_Valve_Blending_DB"."AV-30.03".QOPEN,
                FB_P_Transfer := "IO Motor MCC Panel Blending_DB"."P-31.01".QRUN,
                Level := "IO Analog Blending_DB"."LT-30.01".QOUT,
                TransfPump_AVSpeed := "IO Motor MCC Panel Blending_DB"."P-31.01".QAct_Speed);
END_REGION

REGION Network 37: T-31_Dose_ChiliAwetan_1
   RUNG wire#powerrail
      I_Contact( "T-20.00_DB".ChiliAwet_1.QDOSERun )
      I_Contact( "T-21.00_DB".ChiliAwet_1.QDOSERun )
      I_Contact( "T-30.00_DB".ChiliAwet_1.QDOSERun )
      Contact( "T-02.01_DB".State.Ready_For_Transfer )
      wire#w1
      Coil( "T-31.00_DB".ChiliAwet_1.ISTART_COND )
   END_RUNG
   RUNG wire#w1
      Contact( "IO_Valve_Blending_DB"."AV-31.09".FB_OPEN )
      Coil( "T-31.00_DB".ChiliAwet_1.V_OPEN )
   END_RUNG
   RUNG wire#w1
      I_Contact( "IO_Valve_Blending_DB"."AV-31.09".FB_OPEN )
      Coil( "T-31.00_DB".ChiliAwet_1.V_CLOSE )
   END_RUNG
   RUNG wire#w1
      Contact( "IO Motor MCC Preparation_DB"."P-02.01".FB_ON )
      Coil( "T-31.00_DB".ChiliAwet_1.P_RUN )
   END_RUNG
   RUNG wire#w1
      I_Contact( "IO Motor MCC Preparation_DB"."P-02.01".FB_ON )
      Coil( "T-31.00_DB".ChiliAwet_1.P_STOP )
   END_RUNG
   // the same network as SCL:
   "T-31.00_DB".ChiliAwet_1.ISTART_COND := NOT "T-20.00_DB".ChiliAwet_1.QDOSERun AND NOT "T-21.00_DB".ChiliAwet_1.QDOSERun AND NOT "T-30.00_DB".ChiliAwet_1.QDOSERun AND "T-02.01_DB".State.Ready_For_Transfer;
   "T-31.00_DB".ChiliAwet_1.V_OPEN := "T-31.00_DB".ChiliAwet_1.ISTART_COND AND "IO_Valve_Blending_DB"."AV-31.09".FB_OPEN;
   "T-31.00_DB".ChiliAwet_1.V_CLOSE := "T-31.00_DB".ChiliAwet_1.ISTART_COND AND NOT "IO_Valve_Blending_DB"."AV-31.09".FB_OPEN;
   "T-31.00_DB".ChiliAwet_1.P_RUN := "T-31.00_DB".ChiliAwet_1.ISTART_COND AND "IO Motor MCC Preparation_DB"."P-02.01".FB_ON;
   "T-31.00_DB".ChiliAwet_1.P_STOP := "T-31.00_DB".ChiliAwet_1.ISTART_COND AND NOT "IO Motor MCC Preparation_DB"."P-02.01".FB_ON;
END_REGION

REGION Network 38: T-31_Dose_ChiliAwetan_2
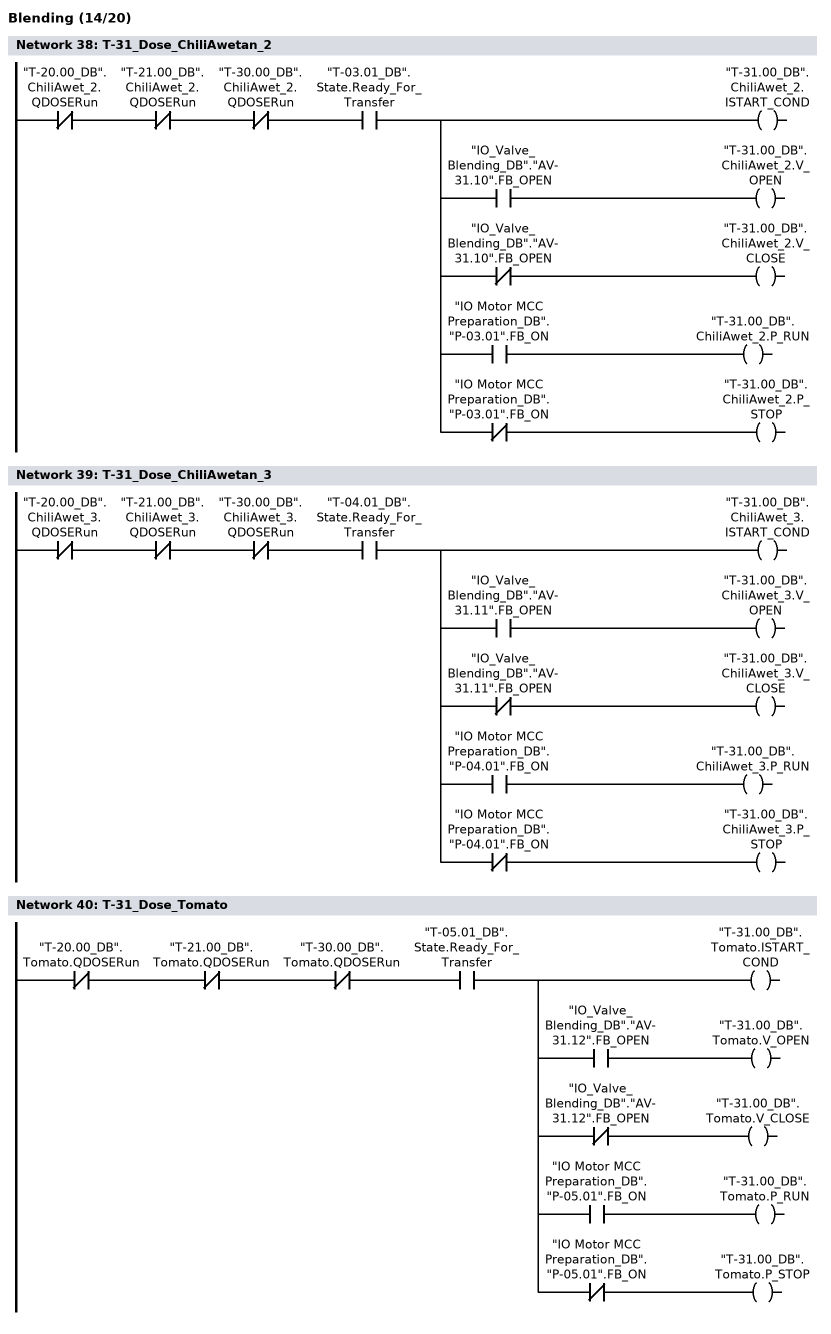
   RUNG wire#powerrail
      I_Contact( "T-20.00_DB".ChiliAwet_2.QDOSERun )
      I_Contact( "T-21.00_DB".ChiliAwet_2.QDOSERun )
      I_Contact( "T-30.00_DB".ChiliAwet_2.QDOSERun )
      Contact( "T-03.01_DB".State.Ready_For_Transfer )
      wire#w1
      Coil( "T-31.00_DB".ChiliAwet_2.ISTART_COND )
   END_RUNG
   RUNG wire#w1
      Contact( "IO_Valve_Blending_DB"."AV-31.10".FB_OPEN )
      Coil( "T-31.00_DB".ChiliAwet_2.V_OPEN )
   END_RUNG
   RUNG wire#w1
      I_Contact( "IO_Valve_Blending_DB"."AV-31.10".FB_OPEN )
      Coil( "T-31.00_DB".ChiliAwet_2.V_CLOSE )
   END_RUNG
   RUNG wire#w1
      Contact( "IO Motor MCC Preparation_DB"."P-03.01".FB_ON )
      Coil( "T-31.00_DB".ChiliAwet_2.P_RUN )
   END_RUNG
   RUNG wire#w1
      I_Contact( "IO Motor MCC Preparation_DB"."P-03.01".FB_ON )
      Coil( "T-31.00_DB".ChiliAwet_2.P_STOP )
   END_RUNG
   // the same network as SCL:
   "T-31.00_DB".ChiliAwet_2.ISTART_COND := NOT "T-20.00_DB".ChiliAwet_2.QDOSERun AND NOT "T-21.00_DB".ChiliAwet_2.QDOSERun AND NOT "T-30.00_DB".ChiliAwet_2.QDOSERun AND "T-03.01_DB".State.Ready_For_Transfer;
   "T-31.00_DB".ChiliAwet_2.V_OPEN := "T-31.00_DB".ChiliAwet_2.ISTART_COND AND "IO_Valve_Blending_DB"."AV-31.10".FB_OPEN;
   "T-31.00_DB".ChiliAwet_2.V_CLOSE := "T-31.00_DB".ChiliAwet_2.ISTART_COND AND NOT "IO_Valve_Blending_DB"."AV-31.10".FB_OPEN;
   "T-31.00_DB".ChiliAwet_2.P_RUN := "T-31.00_DB".ChiliAwet_2.ISTART_COND AND "IO Motor MCC Preparation_DB"."P-03.01".FB_ON;
   "T-31.00_DB".ChiliAwet_2.P_STOP := "T-31.00_DB".ChiliAwet_2.ISTART_COND AND NOT "IO Motor MCC Preparation_DB"."P-03.01".FB_ON;
END_REGION

REGION Network 39: T-31_Dose_ChiliAwetan_3
   RUNG wire#powerrail
      I_Contact( "T-20.00_DB".ChiliAwet_3.QDOSERun )
      I_Contact( "T-21.00_DB".ChiliAwet_3.QDOSERun )
      I_Contact( "T-30.00_DB".ChiliAwet_3.QDOSERun )
      Contact( "T-04.01_DB".State.Ready_For_Transfer )
      wire#w1
      Coil( "T-31.00_DB".ChiliAwet_3.ISTART_COND )
   END_RUNG
   RUNG wire#w1
      Contact( "IO_Valve_Blending_DB"."AV-31.11".FB_OPEN )
      Coil( "T-31.00_DB".ChiliAwet_3.V_OPEN )
   END_RUNG
   RUNG wire#w1
      I_Contact( "IO_Valve_Blending_DB"."AV-31.11".FB_OPEN )
      Coil( "T-31.00_DB".ChiliAwet_3.V_CLOSE )
   END_RUNG
   RUNG wire#w1
      Contact( "IO Motor MCC Preparation_DB"."P-04.01".FB_ON )
      Coil( "T-31.00_DB".ChiliAwet_3.P_RUN )
   END_RUNG
   RUNG wire#w1
      I_Contact( "IO Motor MCC Preparation_DB"."P-04.01".FB_ON )
      Coil( "T-31.00_DB".ChiliAwet_3.P_STOP )
   END_RUNG
   // the same network as SCL:
   "T-31.00_DB".ChiliAwet_3.ISTART_COND := NOT "T-20.00_DB".ChiliAwet_3.QDOSERun AND NOT "T-21.00_DB".ChiliAwet_3.QDOSERun AND NOT "T-30.00_DB".ChiliAwet_3.QDOSERun AND "T-04.01_DB".State.Ready_For_Transfer;
   "T-31.00_DB".ChiliAwet_3.V_OPEN := "T-31.00_DB".ChiliAwet_3.ISTART_COND AND "IO_Valve_Blending_DB"."AV-31.11".FB_OPEN;
   "T-31.00_DB".ChiliAwet_3.V_CLOSE := "T-31.00_DB".ChiliAwet_3.ISTART_COND AND NOT "IO_Valve_Blending_DB"."AV-31.11".FB_OPEN;
   "T-31.00_DB".ChiliAwet_3.P_RUN := "T-31.00_DB".ChiliAwet_3.ISTART_COND AND "IO Motor MCC Preparation_DB"."P-04.01".FB_ON;
   "T-31.00_DB".ChiliAwet_3.P_STOP := "T-31.00_DB".ChiliAwet_3.ISTART_COND AND NOT "IO Motor MCC Preparation_DB"."P-04.01".FB_ON;
END_REGION

REGION Network 40: T-31_Dose_Tomato
   RUNG wire#powerrail
      I_Contact( "T-20.00_DB".Tomato.QDOSERun )
      I_Contact( "T-21.00_DB".Tomato.QDOSERun )
      I_Contact( "T-30.00_DB".Tomato.QDOSERun )
      Contact( "T-05.01_DB".State.Ready_For_Transfer )
      wire#w1
      Coil( "T-31.00_DB".Tomato.ISTART_COND )
   END_RUNG
   RUNG wire#w1
      Contact( "IO_Valve_Blending_DB"."AV-31.12".FB_OPEN )
      Coil( "T-31.00_DB".Tomato.V_OPEN )
   END_RUNG
   RUNG wire#w1
      I_Contact( "IO_Valve_Blending_DB"."AV-31.12".FB_OPEN )
      Coil( "T-31.00_DB".Tomato.V_CLOSE )
   END_RUNG
   RUNG wire#w1
      Contact( "IO Motor MCC Preparation_DB"."P-05.01".FB_ON )
      Coil( "T-31.00_DB".Tomato.P_RUN )
   END_RUNG
   RUNG wire#w1
      I_Contact( "IO Motor MCC Preparation_DB"."P-05.01".FB_ON )
      Coil( "T-31.00_DB".Tomato.P_STOP )
   END_RUNG
   // the same network as SCL:
   "T-31.00_DB".Tomato.ISTART_COND := NOT "T-20.00_DB".Tomato.QDOSERun AND NOT "T-21.00_DB".Tomato.QDOSERun AND NOT "T-30.00_DB".Tomato.QDOSERun AND "T-05.01_DB".State.Ready_For_Transfer;
   "T-31.00_DB".Tomato.V_OPEN := "T-31.00_DB".Tomato.ISTART_COND AND "IO_Valve_Blending_DB"."AV-31.12".FB_OPEN;
   "T-31.00_DB".Tomato.V_CLOSE := "T-31.00_DB".Tomato.ISTART_COND AND NOT "IO_Valve_Blending_DB"."AV-31.12".FB_OPEN;
   "T-31.00_DB".Tomato.P_RUN := "T-31.00_DB".Tomato.ISTART_COND AND "IO Motor MCC Preparation_DB"."P-05.01".FB_ON;
   "T-31.00_DB".Tomato.P_STOP := "T-31.00_DB".Tomato.ISTART_COND AND NOT "IO Motor MCC Preparation_DB"."P-05.01".FB_ON;
END_REGION

REGION Network 41: T-31_Dose_FreshChili_1
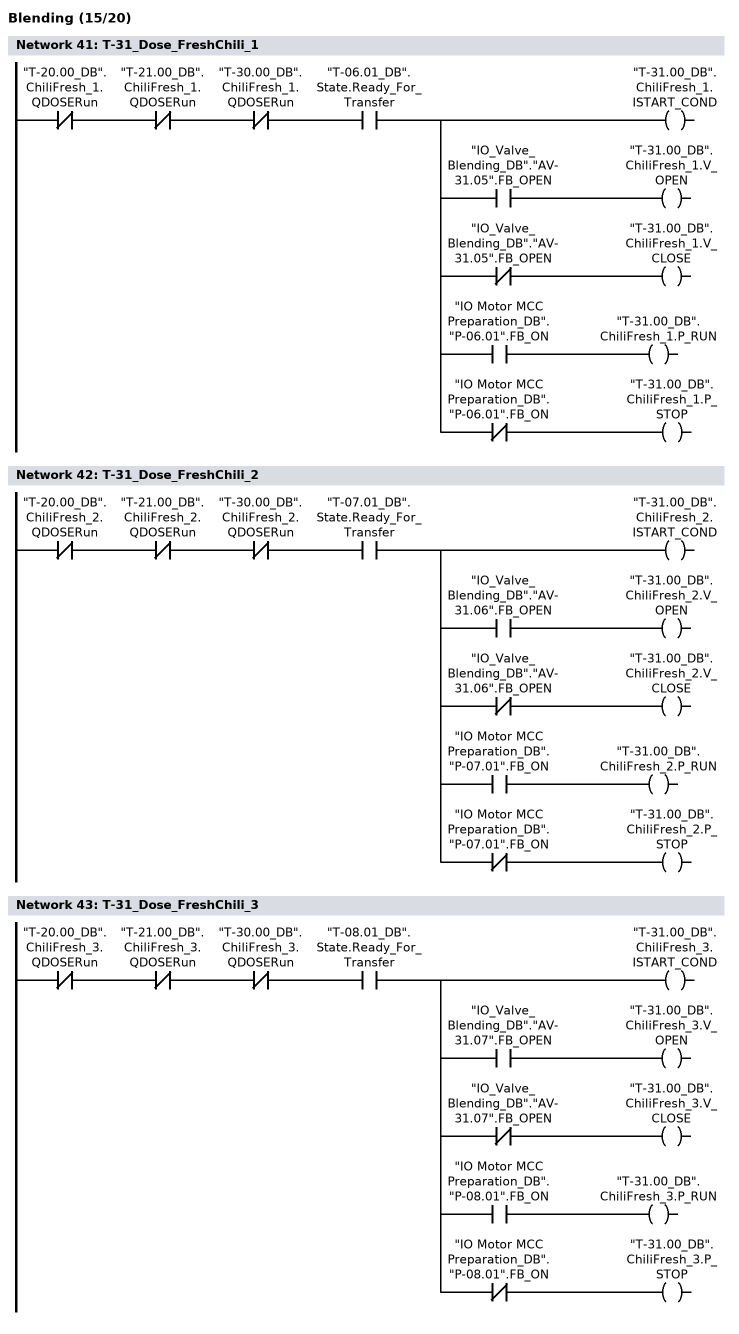
   RUNG wire#powerrail
      I_Contact( "T-20.00_DB".ChiliFresh_1.QDOSERun )
      I_Contact( "T-21.00_DB".ChiliFresh_1.QDOSERun )
      I_Contact( "T-30.00_DB".ChiliFresh_1.QDOSERun )
      Contact( "T-06.01_DB".State.Ready_For_Transfer )
      wire#w1
      Coil( "T-31.00_DB".ChiliFresh_1.ISTART_COND )
   END_RUNG
   RUNG wire#w1
      Contact( "IO_Valve_Blending_DB"."AV-31.05".FB_OPEN )
      Coil( "T-31.00_DB".ChiliFresh_1.V_OPEN )
   END_RUNG
   RUNG wire#w1
      I_Contact( "IO_Valve_Blending_DB"."AV-31.05".FB_OPEN )
      Coil( "T-31.00_DB".ChiliFresh_1.V_CLOSE )
   END_RUNG
   RUNG wire#w1
      Contact( "IO Motor MCC Preparation_DB"."P-06.01".FB_ON )
      Coil( "T-31.00_DB".ChiliFresh_1.P_RUN )
   END_RUNG
   RUNG wire#w1
      I_Contact( "IO Motor MCC Preparation_DB"."P-06.01".FB_ON )
      Coil( "T-31.00_DB".ChiliFresh_1.P_STOP )
   END_RUNG
   // the same network as SCL:
   "T-31.00_DB".ChiliFresh_1.ISTART_COND := NOT "T-20.00_DB".ChiliFresh_1.QDOSERun AND NOT "T-21.00_DB".ChiliFresh_1.QDOSERun AND NOT "T-30.00_DB".ChiliFresh_1.QDOSERun AND "T-06.01_DB".State.Ready_For_Transfer;
   "T-31.00_DB".ChiliFresh_1.V_OPEN := "T-31.00_DB".ChiliFresh_1.ISTART_COND AND "IO_Valve_Blending_DB"."AV-31.05".FB_OPEN;
   "T-31.00_DB".ChiliFresh_1.V_CLOSE := "T-31.00_DB".ChiliFresh_1.ISTART_COND AND NOT "IO_Valve_Blending_DB"."AV-31.05".FB_OPEN;
   "T-31.00_DB".ChiliFresh_1.P_RUN := "T-31.00_DB".ChiliFresh_1.ISTART_COND AND "IO Motor MCC Preparation_DB"."P-06.01".FB_ON;
   "T-31.00_DB".ChiliFresh_1.P_STOP := "T-31.00_DB".ChiliFresh_1.ISTART_COND AND NOT "IO Motor MCC Preparation_DB"."P-06.01".FB_ON;
END_REGION

REGION Network 42: T-31_Dose_FreshChili_2
   RUNG wire#powerrail
      I_Contact( "T-20.00_DB".ChiliFresh_2.QDOSERun )
      I_Contact( "T-21.00_DB".ChiliFresh_2.QDOSERun )
      I_Contact( "T-30.00_DB".ChiliFresh_2.QDOSERun )
      Contact( "T-07.01_DB".State.Ready_For_Transfer )
      wire#w1
      Coil( "T-31.00_DB".ChiliFresh_2.ISTART_COND )
   END_RUNG
   RUNG wire#w1
      Contact( "IO_Valve_Blending_DB"."AV-31.06".FB_OPEN )
      Coil( "T-31.00_DB".ChiliFresh_2.V_OPEN )
   END_RUNG
   RUNG wire#w1
      I_Contact( "IO_Valve_Blending_DB"."AV-31.06".FB_OPEN )
      Coil( "T-31.00_DB".ChiliFresh_2.V_CLOSE )
   END_RUNG
   RUNG wire#w1
      Contact( "IO Motor MCC Preparation_DB"."P-07.01".FB_ON )
      Coil( "T-31.00_DB".ChiliFresh_2.P_RUN )
   END_RUNG
   RUNG wire#w1
      I_Contact( "IO Motor MCC Preparation_DB"."P-07.01".FB_ON )
      Coil( "T-31.00_DB".ChiliFresh_2.P_STOP )
   END_RUNG
   // the same network as SCL:
   "T-31.00_DB".ChiliFresh_2.ISTART_COND := NOT "T-20.00_DB".ChiliFresh_2.QDOSERun AND NOT "T-21.00_DB".ChiliFresh_2.QDOSERun AND NOT "T-30.00_DB".ChiliFresh_2.QDOSERun AND "T-07.01_DB".State.Ready_For_Transfer;
   "T-31.00_DB".ChiliFresh_2.V_OPEN := "T-31.00_DB".ChiliFresh_2.ISTART_COND AND "IO_Valve_Blending_DB"."AV-31.06".FB_OPEN;
   "T-31.00_DB".ChiliFresh_2.V_CLOSE := "T-31.00_DB".ChiliFresh_2.ISTART_COND AND NOT "IO_Valve_Blending_DB"."AV-31.06".FB_OPEN;
   "T-31.00_DB".ChiliFresh_2.P_RUN := "T-31.00_DB".ChiliFresh_2.ISTART_COND AND "IO Motor MCC Preparation_DB"."P-07.01".FB_ON;
   "T-31.00_DB".ChiliFresh_2.P_STOP := "T-31.00_DB".ChiliFresh_2.ISTART_COND AND NOT "IO Motor MCC Preparation_DB"."P-07.01".FB_ON;
END_REGION

REGION Network 43: T-31_Dose_FreshChili_3
   RUNG wire#powerrail
      I_Contact( "T-20.00_DB".ChiliFresh_3.QDOSERun )
      I_Contact( "T-21.00_DB".ChiliFresh_3.QDOSERun )
      I_Contact( "T-30.00_DB".ChiliFresh_3.QDOSERun )
      Contact( "T-08.01_DB".State.Ready_For_Transfer )
      wire#w1
      Coil( "T-31.00_DB".ChiliFresh_3.ISTART_COND )
   END_RUNG
   RUNG wire#w1
      Contact( "IO_Valve_Blending_DB"."AV-31.07".FB_OPEN )
      Coil( "T-31.00_DB".ChiliFresh_3.V_OPEN )
   END_RUNG
   RUNG wire#w1
      I_Contact( "IO_Valve_Blending_DB"."AV-31.07".FB_OPEN )
      Coil( "T-31.00_DB".ChiliFresh_3.V_CLOSE )
   END_RUNG
   RUNG wire#w1
      Contact( "IO Motor MCC Preparation_DB"."P-08.01".FB_ON )
      Coil( "T-31.00_DB".ChiliFresh_3.P_RUN )
   END_RUNG
   RUNG wire#w1
      I_Contact( "IO Motor MCC Preparation_DB"."P-08.01".FB_ON )
      Coil( "T-31.00_DB".ChiliFresh_3.P_STOP )
   END_RUNG
   // the same network as SCL:
   "T-31.00_DB".ChiliFresh_3.ISTART_COND := NOT "T-20.00_DB".ChiliFresh_3.QDOSERun AND NOT "T-21.00_DB".ChiliFresh_3.QDOSERun AND NOT "T-30.00_DB".ChiliFresh_3.QDOSERun AND "T-08.01_DB".State.Ready_For_Transfer;
   "T-31.00_DB".ChiliFresh_3.V_OPEN := "T-31.00_DB".ChiliFresh_3.ISTART_COND AND "IO_Valve_Blending_DB"."AV-31.07".FB_OPEN;
   "T-31.00_DB".ChiliFresh_3.V_CLOSE := "T-31.00_DB".ChiliFresh_3.ISTART_COND AND NOT "IO_Valve_Blending_DB"."AV-31.07".FB_OPEN;
   "T-31.00_DB".ChiliFresh_3.P_RUN := "T-31.00_DB".ChiliFresh_3.ISTART_COND AND "IO Motor MCC Preparation_DB"."P-08.01".FB_ON;
   "T-31.00_DB".ChiliFresh_3.P_STOP := "T-31.00_DB".ChiliFresh_3.ISTART_COND AND NOT "IO Motor MCC Preparation_DB"."P-08.01".FB_ON;
END_REGION

REGION Network 44: T-31_Dose_Garlic
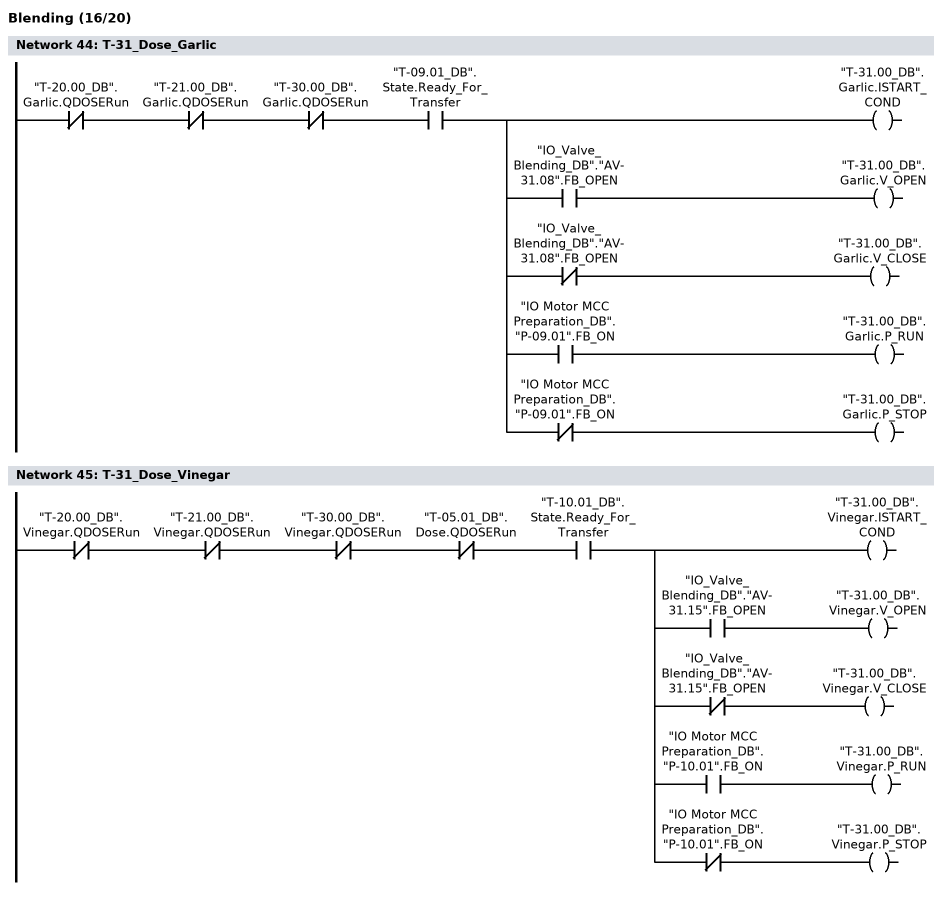
   RUNG wire#powerrail
      I_Contact( "T-20.00_DB".Garlic.QDOSERun )
      I_Contact( "T-21.00_DB".Garlic.QDOSERun )
      I_Contact( "T-30.00_DB".Garlic.QDOSERun )
      Contact( "T-09.01_DB".State.Ready_For_Transfer )
      wire#w1
      Coil( "T-31.00_DB".Garlic.ISTART_COND )
   END_RUNG
   RUNG wire#w1
      Contact( "IO_Valve_Blending_DB"."AV-31.08".FB_OPEN )
      Coil( "T-31.00_DB".Garlic.V_OPEN )
   END_RUNG
   RUNG wire#w1
      I_Contact( "IO_Valve_Blending_DB"."AV-31.08".FB_OPEN )
      Coil( "T-31.00_DB".Garlic.V_CLOSE )
   END_RUNG
   RUNG wire#w1
      Contact( "IO Motor MCC Preparation_DB"."P-09.01".FB_ON )
      Coil( "T-31.00_DB".Garlic.P_RUN )
   END_RUNG
   RUNG wire#w1
      I_Contact( "IO Motor MCC Preparation_DB"."P-09.01".FB_ON )
      Coil( "T-31.00_DB".Garlic.P_STOP )
   END_RUNG
   // the same network as SCL:
   "T-31.00_DB".Garlic.ISTART_COND := NOT "T-20.00_DB".Garlic.QDOSERun AND NOT "T-21.00_DB".Garlic.QDOSERun AND NOT "T-30.00_DB".Garlic.QDOSERun AND "T-09.01_DB".State.Ready_For_Transfer;
   "T-31.00_DB".Garlic.V_OPEN := "T-31.00_DB".Garlic.ISTART_COND AND "IO_Valve_Blending_DB"."AV-31.08".FB_OPEN;
   "T-31.00_DB".Garlic.V_CLOSE := "T-31.00_DB".Garlic.ISTART_COND AND NOT "IO_Valve_Blending_DB"."AV-31.08".FB_OPEN;
   "T-31.00_DB".Garlic.P_RUN := "T-31.00_DB".Garlic.ISTART_COND AND "IO Motor MCC Preparation_DB"."P-09.01".FB_ON;
   "T-31.00_DB".Garlic.P_STOP := "T-31.00_DB".Garlic.ISTART_COND AND NOT "IO Motor MCC Preparation_DB"."P-09.01".FB_ON;
END_REGION

REGION Network 45: T-31_Dose_Vinegar
   RUNG wire#powerrail
      I_Contact( "T-20.00_DB".Vinegar.QDOSERun )
      I_Contact( "T-21.00_DB".Vinegar.QDOSERun )
      I_Contact( "T-30.00_DB".Vinegar.QDOSERun )
      I_Contact( "T-05.01_DB".Dose.QDOSERun )
      Contact( "T-10.01_DB".State.Ready_For_Transfer )
      wire#w1
      Coil( "T-31.00_DB".Vinegar.ISTART_COND )
   END_RUNG
   RUNG wire#w1
      Contact( "IO_Valve_Blending_DB"."AV-31.15".FB_OPEN )
      Coil( "T-31.00_DB".Vinegar.V_OPEN )
   END_RUNG
   RUNG wire#w1
      I_Contact( "IO_Valve_Blending_DB"."AV-31.15".FB_OPEN )
      Coil( "T-31.00_DB".Vinegar.V_CLOSE )
   END_RUNG
   RUNG wire#w1
      Contact( "IO Motor MCC Preparation_DB"."P-10.01".FB_ON )
      Coil( "T-31.00_DB".Vinegar.P_RUN )
   END_RUNG
   RUNG wire#w1
      I_Contact( "IO Motor MCC Preparation_DB"."P-10.01".FB_ON )
      Coil( "T-31.00_DB".Vinegar.P_STOP )
   END_RUNG
   // the same network as SCL:
   "T-31.00_DB".Vinegar.ISTART_COND := NOT "T-20.00_DB".Vinegar.QDOSERun AND NOT "T-21.00_DB".Vinegar.QDOSERun AND NOT "T-30.00_DB".Vinegar.QDOSERun AND NOT "T-05.01_DB".Dose.QDOSERun AND "T-10.01_DB".State.Ready_For_Transfer;
   "T-31.00_DB".Vinegar.V_OPEN := "T-31.00_DB".Vinegar.ISTART_COND AND "IO_Valve_Blending_DB"."AV-31.15".FB_OPEN;
   "T-31.00_DB".Vinegar.V_CLOSE := "T-31.00_DB".Vinegar.ISTART_COND AND NOT "IO_Valve_Blending_DB"."AV-31.15".FB_OPEN;
   "T-31.00_DB".Vinegar.P_RUN := "T-31.00_DB".Vinegar.ISTART_COND AND "IO Motor MCC Preparation_DB"."P-10.01".FB_ON;
   "T-31.00_DB".Vinegar.P_STOP := "T-31.00_DB".Vinegar.ISTART_COND AND NOT "IO Motor MCC Preparation_DB"."P-10.01".FB_ON;
END_REGION

REGION Network 46: T-31.00
   // "IO Analog Blending_DB"."LT-31.01".QOUT
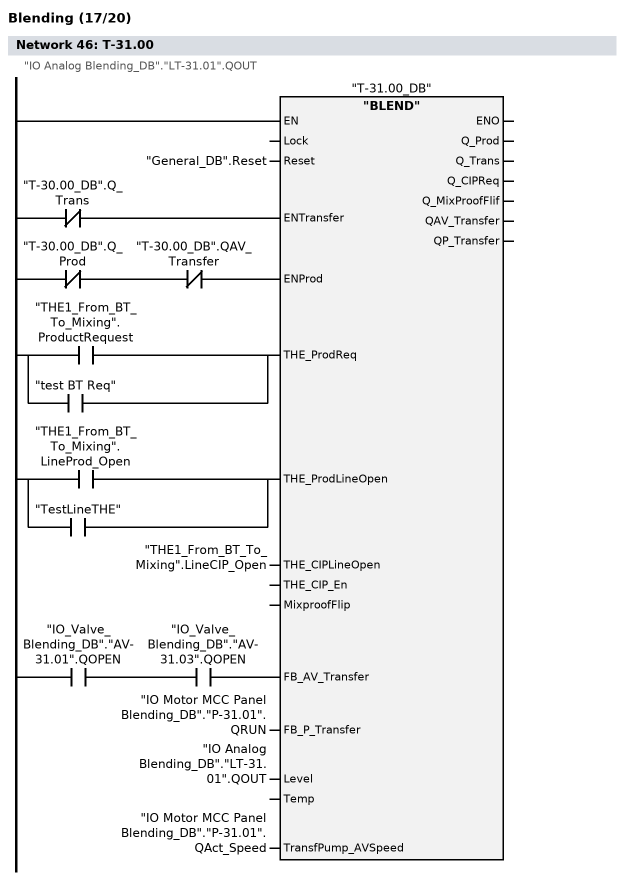
   RUNG wire#powerrail
      "T-31.00_DB"(ENTransfer := wire#w1, ENProd := wire#w2, THE_ProdReq := wire#w3, THE_ProdLineOpen := wire#w4, FB_AV_Transfer := wire#w5, Lock :=, Reset := "General_DB".Reset, THE_CIPLineOpen := "THE1_From_BT_To_Mixing".LineCIP_Open, THE_CIP_En :=, MixproofFlip :=, FB_P_Transfer := "IO Motor MCC Panel Blending_DB"."P-31.01".QRUN, Level := "IO Analog Blending_DB"."LT-31.01".QOUT, Temp :=, TransfPump_AVSpeed := "IO Motor MCC Panel Blending_DB"."P-31.01".QAct_Speed, Q_Prod =>, Q_Trans =>, Q_CIPReq =>, Q_MixProofFlif =>, QAV_Transfer =>, QP_Transfer =>)
   END_RUNG
   RUNG wire#powerrail
      I_Contact( "T-30.00_DB".Q_Trans )
   END_RUNG wire#w1
   RUNG wire#powerrail
      I_Contact( "T-30.00_DB".Q_Prod )
      I_Contact( "T-30.00_DB".QAV_Transfer )
   END_RUNG wire#w2
   RUNG wire#powerrail
      Contact( "THE1_From_BT_To_Mixing".ProductRequest )
   END_RUNG wire#w3
   RUNG wire#powerrail
      Contact( "test BT Req" )
   END_RUNG wire#w3
   RUNG wire#powerrail
      Contact( "THE1_From_BT_To_Mixing".LineProd_Open )
   END_RUNG wire#w4
   RUNG wire#powerrail
      Contact( "TestLineTHE" )
   END_RUNG wire#w4
   RUNG wire#powerrail
      Contact( "IO_Valve_Blending_DB"."AV-31.01".QOPEN )
      Contact( "IO_Valve_Blending_DB"."AV-31.03".QOPEN )
   END_RUNG wire#w5
   // the same network as SCL:
   "T-31.00_DB"(Reset := "General_DB".Reset,   // "BLEND"
                ENTransfer := NOT "T-30.00_DB".Q_Trans,
                ENProd := NOT "T-30.00_DB".Q_Prod AND NOT "T-30.00_DB".QAV_Transfer,
                THE_ProdReq := "THE1_From_BT_To_Mixing".ProductRequest OR "test BT Req",
                THE_ProdLineOpen := "THE1_From_BT_To_Mixing".LineProd_Open OR "TestLineTHE",
                THE_CIPLineOpen := "THE1_From_BT_To_Mixing".LineCIP_Open,
                FB_AV_Transfer := "IO_Valve_Blending_DB"."AV-31.01".QOPEN AND "IO_Valve_Blending_DB"."AV-31.03".QOPEN,
                FB_P_Transfer := "IO Motor MCC Panel Blending_DB"."P-31.01".QRUN,
                Level := "IO Analog Blending_DB"."LT-31.01".QOUT,
                TransfPump_AVSpeed := "IO Motor MCC Panel Blending_DB"."P-31.01".QAct_Speed);
END_REGION

REGION Network 47: Comm to Buffer Tank THE 1
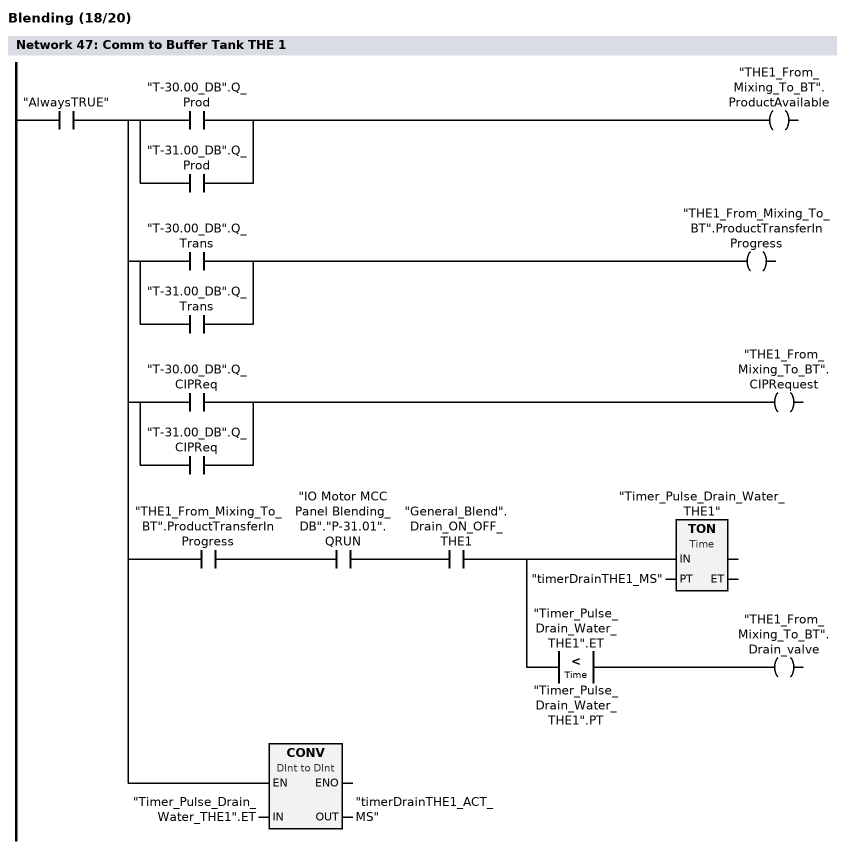
   RUNG wire#powerrail
      Contact( "AlwaysTRUE" )
      wire#w1
      Contact( "T-30.00_DB".Q_Prod )
      wire#w2
      Coil( "THE1_From_Mixing_To_BT".ProductAvailable )
   END_RUNG
   RUNG wire#w1
      Contact( "T-31.00_DB".Q_Prod )
   END_RUNG wire#w2
   RUNG wire#w1
      Contact( "T-30.00_DB".Q_Trans )
      wire#w3
      Coil( "THE1_From_Mixing_To_BT".ProductTransferInProgress )
   END_RUNG
   RUNG wire#w1
      Contact( "T-31.00_DB".Q_Trans )
   END_RUNG wire#w3
   RUNG wire#w1
      Contact( "T-30.00_DB".Q_CIPReq )
      wire#w4
      Coil( "THE1_From_Mixing_To_BT".CIPRequest )
   END_RUNG
   RUNG wire#w1
      Contact( "T-31.00_DB".Q_CIPReq )
   END_RUNG wire#w4
   RUNG wire#w1
      Contact( "THE1_From_Mixing_To_BT".ProductTransferInProgress )
      Contact( "IO Motor MCC Panel Blending_DB"."P-31.01".QRUN )
      Contact( "General_Blend".Drain_ON_OFF_THE1 )
      wire#w5
      { S7_Templates := "time_type := Time" } "Timer_Pulse_Drain_Water_THE1".TON(pt := "timerDrainTHE1_MS", et =>)
   END_RUNG
   RUNG wire#w5
      { S7_Templates := "SrcType := Time" } LT_Contact(in1 := "Timer_Pulse_Drain_Water_THE1".ET, in2 := "Timer_Pulse_Drain_Water_THE1".PT)
      Coil( "THE1_From_Mixing_To_BT".Drain_valve )
   END_RUNG
   RUNG wire#w1
      { S7_Templates := "[SrcType := DInt, DestType := DInt]" } Convert(in := "Timer_Pulse_Drain_Water_THE1".ET, out => "timerDrainTHE1_ACT_MS")
   END_RUNG
   // the same network as SCL:
   "THE1_From_Mixing_To_BT".ProductAvailable := "AlwaysTRUE" AND ("T-30.00_DB".Q_Prod OR "T-31.00_DB".Q_Prod);
   "THE1_From_Mixing_To_BT".ProductTransferInProgress := "AlwaysTRUE" AND ("T-30.00_DB".Q_Trans OR "T-31.00_DB".Q_Trans);
   "THE1_From_Mixing_To_BT".CIPRequest := "AlwaysTRUE" AND ("T-30.00_DB".Q_CIPReq OR "T-31.00_DB".Q_CIPReq);
   #_w1 := "AlwaysTRUE" AND "THE1_From_Mixing_To_BT".ProductTransferInProgress AND "IO Motor MCC Panel Blending_DB"."P-31.01".QRUN AND "General_Blend".Drain_ON_OFF_THE1;
   "Timer_Pulse_Drain_Water_THE1".TON(IN := #_w1, PT := "timerDrainTHE1_MS");
   "THE1_From_Mixing_To_BT".Drain_valve := #_w1 AND ("Timer_Pulse_Drain_Water_THE1".ET < "Timer_Pulse_Drain_Water_THE1".PT);
   IF "AlwaysTRUE" THEN "timerDrainTHE1_ACT_MS" := DINT_TO_DINT("Timer_Pulse_Drain_Water_THE1".ET); END_IF;
END_REGION

REGION Network 48: Rework T-22
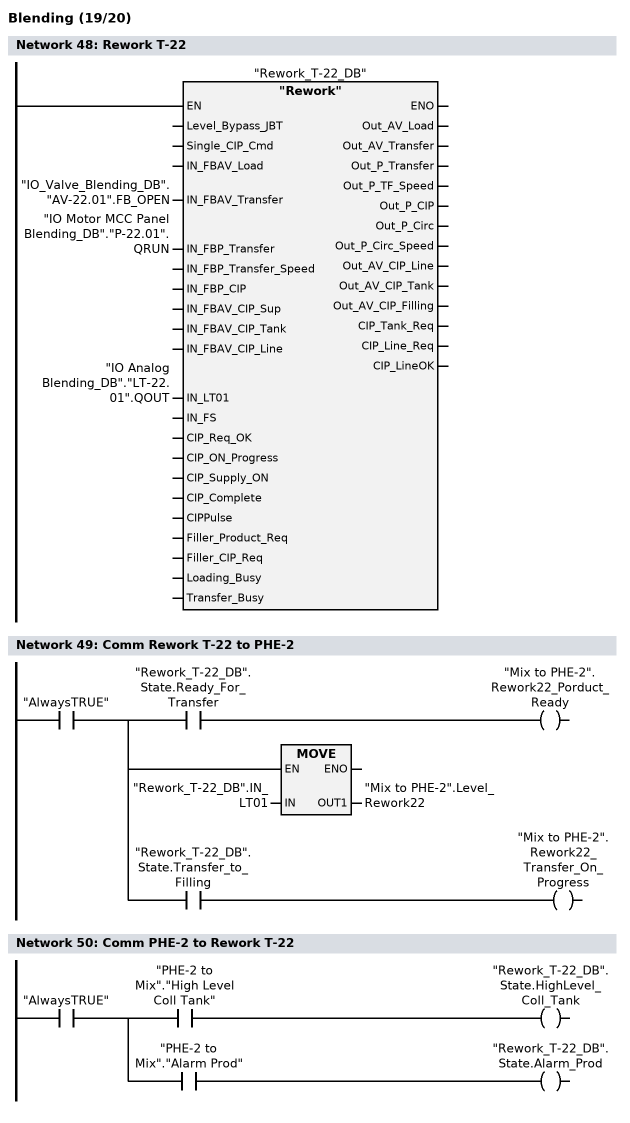
   RUNG wire#powerrail
      "Rework_T-22_DB"(Level_Bypass_JBT :=, Single_CIP_Cmd :=, IN_FBAV_Load :=, IN_FBAV_Transfer := "IO_Valve_Blending_DB"."AV-22.01".FB_OPEN, IN_FBP_Transfer := "IO Motor MCC Panel Blending_DB"."P-22.01".QRUN, IN_FBP_Transfer_Speed :=, IN_FBP_CIP :=, IN_FBAV_CIP_Sup :=, IN_FBAV_CIP_Tank :=, IN_FBAV_CIP_Line :=, IN_LT01 := "IO Analog Blending_DB"."LT-22.01".QOUT, IN_FS :=, CIP_Req_OK :=, CIP_ON_Progress :=, CIP_Supply_ON :=, CIP_Complete :=, CIPPulse :=, Filler_Product_Req :=, Filler_CIP_Req :=, Loading_Busy :=, Transfer_Busy :=, Out_AV_Load =>, Out_AV_Transfer =>, Out_P_Transfer =>, Out_P_TF_Speed =>, Out_P_CIP =>, Out_P_Circ =>, Out_P_Circ_Speed =>, Out_AV_CIP_Line =>, Out_AV_CIP_Tank =>, Out_AV_CIP_Filling =>, CIP_Tank_Req =>, CIP_Line_Req =>, CIP_LineOK =>)
   END_RUNG
   // the same network as SCL:
   "Rework_T-22_DB"(IN_FBAV_Transfer := "IO_Valve_Blending_DB"."AV-22.01".FB_OPEN,   // "Rework"
                    IN_FBP_Transfer := "IO Motor MCC Panel Blending_DB"."P-22.01".QRUN,
                    IN_LT01 := "IO Analog Blending_DB"."LT-22.01".QOUT);
END_REGION

REGION Network 49: Comm Rework T-22 to PHE-2
   RUNG wire#powerrail
      Contact( "AlwaysTRUE" )
      wire#w1
      Contact( "Rework_T-22_DB".State.Ready_For_Transfer )
      Coil( "Mix to PHE-2".Rework22_Porduct_Ready )
   END_RUNG
   RUNG wire#w1
      Move(in := "Rework_T-22_DB".IN_LT01, out1 => "Mix to PHE-2".Level_Rework22)
   END_RUNG
   RUNG wire#w1
      Contact( "Rework_T-22_DB".State.Transfer_to_Filling )
      Coil( "Mix to PHE-2".Rework22_Transfer_On_Progress )
   END_RUNG
   // the same network as SCL:
   "Mix to PHE-2".Rework22_Porduct_Ready := "AlwaysTRUE" AND "Rework_T-22_DB".State.Ready_For_Transfer;
   IF "AlwaysTRUE" THEN "Mix to PHE-2".Level_Rework22 := "Rework_T-22_DB".IN_LT01; END_IF;
   "Mix to PHE-2".Rework22_Transfer_On_Progress := "AlwaysTRUE" AND "Rework_T-22_DB".State.Transfer_to_Filling;
END_REGION

REGION Network 50: Comm PHE-2 to Rework T-22
   RUNG wire#powerrail
      Contact( "AlwaysTRUE" )
      wire#w1
      Contact( "PHE-2 to Mix"."High Level Coll Tank" )
      Coil( "Rework_T-22_DB".State.HighLevel_Coll_Tank )
   END_RUNG
   RUNG wire#w1
      Contact( "PHE-2 to Mix"."Alarm Prod" )
      Coil( "Rework_T-22_DB".State.Alarm_Prod )
   END_RUNG
   // the same network as SCL:
   "Rework_T-22_DB".State.HighLevel_Coll_Tank := "AlwaysTRUE" AND "PHE-2 to Mix"."High Level Coll Tank";
   "Rework_T-22_DB".State.Alarm_Prod := "AlwaysTRUE" AND "PHE-2 to Mix"."Alarm Prod";
END_REGION

REGION Network 51: Rework T-32
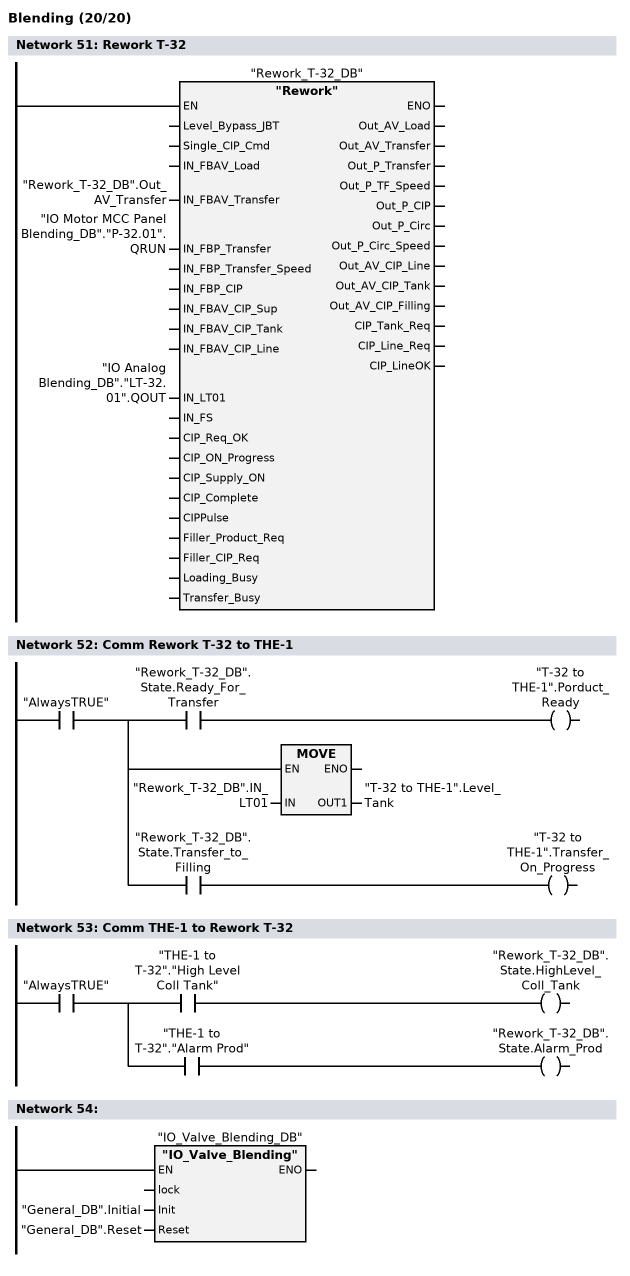
   RUNG wire#powerrail
      "Rework_T-32_DB"(Level_Bypass_JBT :=, Single_CIP_Cmd :=, IN_FBAV_Load :=, IN_FBAV_Transfer := "Rework_T-32_DB".Out_AV_Transfer, IN_FBP_Transfer := "IO Motor MCC Panel Blending_DB"."P-32.01".QRUN, IN_FBP_Transfer_Speed :=, IN_FBP_CIP :=, IN_FBAV_CIP_Sup :=, IN_FBAV_CIP_Tank :=, IN_FBAV_CIP_Line :=, IN_LT01 := "IO Analog Blending_DB"."LT-32.01".QOUT, IN_FS :=, CIP_Req_OK :=, CIP_ON_Progress :=, CIP_Supply_ON :=, CIP_Complete :=, CIPPulse :=, Filler_Product_Req :=, Filler_CIP_Req :=, Loading_Busy :=, Transfer_Busy :=, Out_AV_Load =>, Out_AV_Transfer =>, Out_P_Transfer =>, Out_P_TF_Speed =>, Out_P_CIP =>, Out_P_Circ =>, Out_P_Circ_Speed =>, Out_AV_CIP_Line =>, Out_AV_CIP_Tank =>, Out_AV_CIP_Filling =>, CIP_Tank_Req =>, CIP_Line_Req =>, CIP_LineOK =>)
   END_RUNG
   // the same network as SCL:
   "Rework_T-32_DB"(IN_FBAV_Transfer := "Rework_T-32_DB".Out_AV_Transfer,   // "Rework"
                    IN_FBP_Transfer := "IO Motor MCC Panel Blending_DB"."P-32.01".QRUN,
                    IN_LT01 := "IO Analog Blending_DB"."LT-32.01".QOUT);
END_REGION

REGION Network 52: Comm Rework T-32 to THE-1
   RUNG wire#powerrail
      Contact( "AlwaysTRUE" )
      wire#w1
      Contact( "Rework_T-32_DB".State.Ready_For_Transfer )
      Coil( "T-32 to THE-1".Porduct_Ready )
   END_RUNG
   RUNG wire#w1
      Move(in := "Rework_T-32_DB".IN_LT01, out1 => "T-32 to THE-1".Level_Tank)
   END_RUNG
   RUNG wire#w1
      Contact( "Rework_T-32_DB".State.Transfer_to_Filling )
      Coil( "T-32 to THE-1".Transfer_On_Progress )
   END_RUNG
   // the same network as SCL:
   "T-32 to THE-1".Porduct_Ready := "AlwaysTRUE" AND "Rework_T-32_DB".State.Ready_For_Transfer;
   IF "AlwaysTRUE" THEN "T-32 to THE-1".Level_Tank := "Rework_T-32_DB".IN_LT01; END_IF;
   "T-32 to THE-1".Transfer_On_Progress := "AlwaysTRUE" AND "Rework_T-32_DB".State.Transfer_to_Filling;
END_REGION

REGION Network 53: Comm THE-1 to Rework T-32
   RUNG wire#powerrail
      Contact( "AlwaysTRUE" )
      wire#w1
      Contact( "THE-1 to T-32"."High Level Coll Tank" )
      Coil( "Rework_T-32_DB".State.HighLevel_Coll_Tank )
   END_RUNG
   RUNG wire#w1
      Contact( "THE-1 to T-32"."Alarm Prod" )
      Coil( "Rework_T-32_DB".State.Alarm_Prod )
   END_RUNG
   // the same network as SCL:
   "Rework_T-32_DB".State.HighLevel_Coll_Tank := "AlwaysTRUE" AND "THE-1 to T-32"."High Level Coll Tank";
   "Rework_T-32_DB".State.Alarm_Prod := "AlwaysTRUE" AND "THE-1 to T-32"."Alarm Prod";
END_REGION

REGION Network 54
   RUNG wire#powerrail
      "IO_Valve_Blending_DB"(lock :=, Init := "General_DB".Initial, Reset := "General_DB".Reset)
   END_RUNG
   // the same network as SCL:
   "IO_Valve_Blending_DB"(Init := "General_DB".Initial, Reset := "General_DB".Reset);   // "IO_Valve_Blending"
END_REGION
END_FUNCTION
